C01814=1058.438,-41.200,-66.868,171.247,28.098,155.263
C01815=1058.445,-40.951,-66.880,171.248,28.101,155.263
C01816=1058.451,-40.701,-66.893,171.250,28.102,155.263
C01817=1058.457,-40.452,-66.906,171.252,28.105,155.263
C01818=1058.463,-40.202,-66.919,171.253,28.106,155.264
C01819=1058.469,-39.952,-66.931,171.255,28.108,155.264
C01820=1058.476,-39.703,-66.944,171.257,28.110,155.264
C01821=1058.482,-39.453,-66.956,171.259,28.112,155.264
C01822=1058.488,-39.204,-66.970,171.260,28.114,155.264
C01823=1058.494,-38.954,-66.982,171.262,28.116,155.265
C01824=1058.500,-38.705,-66.996,171.264,28.117,155.265
C01825=1058.507,-38.454,-67.008,171.265,28.120,155.265
C01826=1058.513,-38.205,-67.022,171.267,28.121,155.265
C01827=1058.519,-37.955,-67.034,171.269,28.124,155.265
C01828=1058.525,-37.706,-67.048,171.270,28.126,155.266
C01829=1058.531,-37.456,-67.060,171.272,28.128,155.266
C01830=1058.537,-37.207,-67.073,171.274,28.130,155.266
C01831=1058.543,-36.957,-67.086,171.275,28.131,155.266
C01832=1058.550,-36.708,-67.099,171.277,28.134,155.266
C01833=1058.555,-36.458,-67.112,171.279,28.135,155.267
C01834=1058.562,-36.208,-67.125,171.279,28.137,155.267
C01835=1058.568,-35.959,-67.138,171.281,28.139,155.267
C01836=1058.574,-35.709,-67.151,171.283,28.141,155.267
C01837=1058.580,-35.460,-67.164,171.284,28.144,155.268
C01838=1058.586,-35.210,-67.177,171.286,28.145,155.268
C01839=1058.592,-34.961,-67.190,171.288,28.147,155.268
C01840=1058.599,-34.682,-67.204,171.290,28.150,155.268
C01841=1058.606,-34.402,-67.220,171.292,28.152,155.268
C01842=1058.613,-34.123,-67.234,171.294,28.154,155.269
C01843=1058.620,-33.844,-67.249,171.295,28.156,155.269
C01844=1058.626,-33.594,-67.261,171.297,28.158,155.269
C01845=1058.632,-33.345,-67.275,171.299,28.160,155.269
C01846=1058.638,-33.096,-67.288,171.301,28.162,155.270
C01847=1058.644,-32.846,-67.300,171.302,28.164,155.270
C01848=1058.650,-32.597,-67.314,171.304,28.166,155.270
C01849=1058.656,-32.346,-67.328,171.306,28.168,155.270
C01850=1058.663,-32.097,-67.341,171.307,28.171,155.271
C01851=1058.669,-31.847,-67.354,171.309,28.172,155.271
C01852=1058.675,-31.598,-67.367,171.311,28.175,155.271
C01853=1058.681,-31.349,-67.380,171.312,28.176,155.271
C01854=1058.687,-31.099,-67.393,171.314,28.178,155.271
C01855=1058.694,-30.849,-67.406,171.316,28.181,155.272
C01856=1058.700,-30.600,-67.420,171.317,28.182,155.272
C01857=1058.706,-30.350,-67.433,171.319,28.185,155.272
C01858=1058.712,-30.101,-67.446,171.321,28.186,155.272
C01859=1058.718,-29.851,-67.459,171.322,28.188,155.272
C01860=1058.724,-29.602,-67.473,171.324,28.191,155.273
C01861=1058.731,-29.352,-67.486,171.326,28.192,155.273
C01862=1058.736,-29.102,-67.499,171.327,28.195,155.273
C01863=1058.743,-28.853,-67.512,171.328,28.197,155.273
C01864=1058.749,-28.603,-67.525,171.330,28.198,155.274
C01865=1058.756,-28.353,-67.539,171.331,28.201,155.274
C01866=1058.762,-28.104,-67.552,171.333,28.203,155.274
C01867=1058.768,-27.855,-67.566,171.335,28.204,155.274
C01868=1058.774,-27.605,-67.578,171.337,28.207,155.275
C01869=1058.780,-27.355,-67.592,171.338,28.209,155.275
C01870=1058.786,-27.105,-67.606,171.340,28.211,155.275
C01871=1058.793,-26.856,-67.619,171.342,28.213,155.275
C01872=1058.799,-26.607,-67.632,171.343,28.215,155.275
C01873=1058.805,-26.358,-67.645,171.345,28.217,155.276
C01874=1058.811,-26.107,-67.660,171.347,28.219,155.276
C01875=1058.817,-25.857,-67.672,171.348,28.221,155.276
C01876=1058.823,-25.608,-67.686,171.350,28.223,155.276
C01877=1058.829,-25.359,-67.699,171.352,28.226,155.277
C01878=1058.835,-25.109,-67.713,171.353,28.227,155.277
C01879=1058.842,-24.859,-67.726,171.355,28.230,155.277
C01880=1058.847,-24.610,-67.740,171.357,28.232,155.277
C01881=1058.853,-24.361,-67.753,171.358,28.234,155.278
C01882=1058.860,-24.111,-67.767,171.360,28.236,155.278
C01883=1058.866,-23.861,-67.781,171.362,28.238,155.278
C01884=1058.872,-23.612,-67.794,171.362,28.240,155.278
C01885=1058.877,-23.362,-67.808,171.364,28.242,155.279
C01886=1058.884,-23.113,-67.821,171.366,28.244,155.279
C01887=1058.890,-22.863,-67.835,171.367,28.247,155.279
C01888=1058.896,-22.613,-67.849,171.369,28.249,155.279
C01889=1058.902,-22.364,-67.862,171.371,28.251,155.280
C01890=1058.908,-22.115,-67.875,171.372,28.253,155.280
C01891=1058.914,-21.865,-67.890,171.374,28.255,155.280
C01892=1058.921,-21.615,-67.903,171.376,28.257,155.280
C01893=1058.927,-21.366,-67.916,171.377,28.260,155.281
C01894=1058.933,-21.116,-67.930,171.379,28.261,155.281
C01895=1058.939,-20.867,-67.944,171.381,28.263,155.281
C01896=1058.945,-20.617,-67.957,171.382,28.266,155.281
C01897=1058.951,-20.368,-67.971,171.384,28.268,155.282
C01898=1058.958,-20.118,-67.984,171.386,28.270,155.282
C01899=1058.963,-19.869,-67.999,171.386,28.272,155.282
C01900=1058.970,-19.619,-68.012,171.388,28.274,155.282
C01901=1058.976,-19.370,-68.026,171.390,28.276,155.283
C01902=1058.982,-19.120,-68.040,171.391,28.278,155.283
C01903=1058.988,-18.871,-68.053,171.393,28.281,155.283
C01904=1058.994,-18.590,-68.068,171.395,28.283,155.283
C01905=1059.002,-18.311,-68.084,171.397,28.286,155.284
C01906=1059.009,-18.031,-68.099,171.399,28.288,155.284
C01907=1059.015,-17.751,-68.115,171.401,28.290,155.284
C01908=1059.022,-17.501,-68.128,171.402,28.293,155.285
C01909=1059.028,-17.252,-68.143,171.404,28.295,155.285
C01910=1059.034,-17.003,-68.156,171.406,28.297,155.285
C01911=1059.040,-16.753,-68.170,171.407,28.299,155.285
C01912=1059.047,-16.503,-68.184,171.409,28.301,155.286
C01913=1059.053,-16.253,-68.197,171.410,28.303,155.286
C01914=1059.059,-16.004,-68.211,171.411,28.305,155.286
C01915=1059.065,-15.755,-68.225,171.413,28.307,155.286
C01916=1059.071,-15.505,-68.239,171.415,28.310,155.287
C01917=1059.078,-15.256,-68.253,171.416,28.312,155.287
C01918=1059.084,-15.005,-68.267,171.418,28.314,155.287
C01919=1059.090,-14.757,-68.281,171.420,28.316,155.287
C01920=1059.096,-14.507,-68.295,171.421,28.319,155.288
C01921=1059.103,-14.257,-68.308,171.423,28.321,155.288
C01922=1059.108,-14.008,-68.323,171.425,28.323,155.288
C01923=1059.114,-13.759,-68.337,171.426,28.325,155.289
C01924=1059.121,-13.509,-68.350,171.428,28.328,155.289
C01925=1059.126,-13.259,-68.364,171.429,28.330,155.289
C01926=1059.133,-13.009,-68.379,171.430,28.332,155.289
C01927=1059.139,-12.760,-68.393,171.432,28.334,155.290
C01928=1059.144,-12.511,-68.406,171.434,28.336,155.290
C01929=1059.151,-12.261,-68.421,171.435,28.339,155.290
C01930=1059.157,-12.012,-68.435,171.437,28.341,155.290
C01931=1059.163,-11.761,-68.449,171.439,28.343,155.291
C01932=1059.169,-11.513,-68.463,171.440,28.345,155.291
C01933=1059.175,-11.263,-68.477,171.442,28.347,155.291
C01934=1059.181,-11.013,-68.492,171.443,28.350,155.292
C01935=1059.187,-10.764,-68.505,171.445,28.352,155.292
C01936=1059.194,-10.514,-68.519,171.446,28.354,155.292
C01937=1059.199,-10.265,-68.534,171.448,28.356,155.292
C01938=1059.206,-10.015,-68.547,171.449,28.358,155.293
C01939=1059.212,-9.766,-68.562,171.451,28.361,155.293
C01940=1059.218,-9.516,-68.576,171.453,28.363,155.293
C01941=1059.224,-9.266,-68.589,171.454,28.365,155.293
C01942=1059.231,-9.017,-68.604,171.456,28.367,155.294
C01943=1059.236,-8.767,-68.618,171.457,28.370,155.294
C01944=1059.243,-8.519,-68.632,171.459,28.372,155.294
C01945=1059.249,-8.268,-68.647,171.461,28.374,155.295
C01946=1059.254,-8.019,-68.661,171.462,28.376,155.295
C01947=1059.261,-7.769,-68.675,171.463,28.378,155.295
C01948=1059.267,-7.520,-68.689,171.465,28.381,155.295
C01949=1059.273,-7.270,-68.704,171.467,28.383,155.296
C01950=1059.279,-7.021,-68.718,171.468,28.386,155.296
C01951=1059.286,-6.771,-68.732,171.470,28.388,155.296
C01952=1059.292,-6.522,-68.746,171.471,28.390,155.297
C01953=1059.298,-6.272,-68.761,171.473,28.392,155.297
C01954=1059.304,-6.023,-68.775,171.475,28.394,155.297
C01955=1059.310,-5.773,-68.789,171.476,28.397,155.297
C01956=1059.317,-5.523,-68.804,171.477,28.399,155.298
C01957=1059.322,-5.274,-68.818,171.479,28.401,155.298
C01958=1059.329,-5.025,-68.832,171.480,28.403,155.298
C01959=1059.335,-4.776,-68.847,171.482,28.405,155.298
C01960=1059.341,-4.525,-68.861,171.484,28.408,155.299
C01961=1059.348,-4.277,-68.875,171.485,28.410,155.299
C01962=1059.354,-4.026,-68.889,171.487,28.412,155.299
C01963=1059.359,-3.777,-68.904,171.489,28.414,155.300
C01964=1059.366,-3.528,-68.918,171.490,28.417,155.300
C01965=1059.373,-3.278,-68.932,171.491,28.419,155.300
C01966=1059.378,-3.029,-68.947,171.493,28.421,155.301
C01967=1059.384,-2.779,-68.961,171.494,28.424,155.301
C01968=1059.391,-2.498,-68.978,171.496,28.426,155.301
C01969=1059.397,-2.216,-68.994,171.498,28.429,155.301
C01970=1059.405,-1.935,-69.010,171.500,28.432,155.302
C01971=1059.411,-1.653,-69.027,171.502,28.435,155.302
C01972=1059.417,-1.403,-69.042,171.503,28.437,155.302
C01973=1059.423,-1.154,-69.056,171.504,28.439,155.303
C01974=1059.429,-0.904,-69.071,171.506,28.441,155.303
C01975=1059.435,-0.655,-69.085,171.507,28.444,155.303
C01976=1059.441,-0.406,-69.100,171.509,28.446,155.304
C01977=1059.447,-0.157,-69.115,171.511,28.448,155.304
C01978=1059.453,0.094,-69.129,171.512,28.450,155.304
C01979=1059.459,0.343,-69.143,171.514,28.453,155.305
C01980=1059.465,0.592,-69.158,171.516,28.456,155.305
C01981=1059.472,0.842,-69.173,171.516,28.458,155.305
C01982=1059.477,1.092,-69.187,171.518,28.460,155.305
C01983=1059.484,1.341,-69.202,171.520,28.463,155.306
C01984=1059.489,1.590,-69.217,171.521,28.465,155.306
C01985=1059.496,1.840,-69.232,171.523,28.467,155.306
C01986=1059.501,2.089,-69.246,171.525,28.469,155.307
C01987=1059.508,2.339,-69.260,171.526,28.472,155.307
C01988=1059.514,2.589,-69.275,171.527,28.474,155.307
C01989=1059.520,2.838,-69.290,171.529,28.476,155.308
C01990=1059.526,3.087,-69.305,171.530,28.478,155.308
C01991=1059.532,3.337,-69.320,171.532,28.481,155.308
C01992=1059.538,3.586,-69.334,171.534,28.484,155.309
C01993=1059.544,3.836,-69.349,171.535,28.486,155.309
C01994=1059.550,4.085,-69.363,171.537,28.489,155.309
C01995=1059.557,4.335,-69.378,171.538,28.491,155.309
C01996=1059.563,4.584,-69.393,171.539,28.493,155.310
C01997=1059.569,4.833,-69.408,171.541,28.495,155.310
C01998=1059.574,5.083,-69.423,171.542,28.498,155.310
C01999=1059.581,5.333,-69.438,171.544,28.500,155.311
C02000=1059.586,5.582,-69.453,171.546,28.502,155.311
C02001=1059.593,5.832,-69.468,171.547,28.504,155.311
C02002=1059.599,6.081,-69.483,171.549,28.507,155.312
C02003=1059.605,6.331,-69.497,171.550,28.509,155.312
C02004=1059.611,6.581,-69.512,171.551,28.512,155.312
C02005=1059.618,6.830,-69.526,171.553,28.514,155.313
C02006=1059.623,7.079,-69.541,171.555,28.517,155.313
C02007=1059.630,7.329,-69.556,171.556,28.519,155.313
C02008=1059.636,7.578,-69.571,171.558,28.521,155.313
C02009=1059.642,7.827,-69.586,171.560,28.524,155.314
C02010=1059.648,8.077,-69.600,171.560,28.526,155.314
C02011=1059.654,8.327,-69.616,171.562,28.528,155.314
C02012=1059.660,8.577,-69.631,171.564,28.530,155.315
C02013=1059.666,8.826,-69.646,171.565,28.533,155.315
C02014=1059.672,9.075,-69.660,171.567,28.535,155.315
C02015=1059.679,9.325,-69.675,171.569,28.537,155.316
C02016=1059.685,9.574,-69.690,171.570,28.540,155.316
C02017=1059.691,9.824,-69.705,171.571,28.542,155.316
C02018=1059.697,10.073,-69.720,171.573,28.544,155.317
C02019=1059.704,10.322,-69.736,171.574,28.547,155.317
C02020=1059.710,10.571,-69.750,171.576,28.550,155.317
C02021=1059.715,10.821,-69.766,171.578,28.552,155.318
C02022=1059.722,11.071,-69.781,171.579,28.554,155.318
C02023=1059.728,11.320,-69.796,171.581,28.556,155.318
C02024=1059.735,11.570,-69.811,171.582,28.559,155.318
C02025=1059.740,11.819,-69.825,171.583,28.561,155.319
C02026=1059.747,12.069,-69.840,171.585,28.563,155.319
C02027=1059.753,12.318,-69.855,171.587,28.566,155.319
C02028=1059.760,12.568,-69.870,171.588,28.568,155.320
C02029=1059.765,12.817,-69.886,171.590,28.570,155.320
C02030=1059.771,13.066,-69.901,171.592,28.573,155.320
C02031=1059.778,13.316,-69.916,171.592,28.575,155.321
C02032=1059.785,13.600,-69.932,171.595,28.578,155.321
C02033=1059.792,13.883,-69.950,171.596,28.580,155.321
C02034=1059.799,14.166,-69.967,171.598,28.583,155.322
C02035=1059.806,14.450,-69.984,171.600,28.586,155.322
C02036=1059.812,14.699,-70.000,171.601,28.588,155.322
C02037=1059.819,14.949,-70.015,171.603,28.591,155.323
C02038=1059.824,15.198,-70.030,171.604,28.593,155.323
C02039=1059.830,15.448,-70.045,171.605,28.595,155.323
C02040=1059.837,15.697,-70.060,171.607,28.598,155.324
C02041=1059.843,15.947,-70.076,171.609,28.600,155.324
C02042=1059.848,16.196,-70.091,171.610,28.603,155.324
C02043=1059.854,16.446,-70.106,171.612,28.605,155.325
C02044=1059.860,16.695,-70.121,171.613,28.607,155.325
C02045=1059.867,16.944,-70.137,171.614,28.610,155.325
C02046=1059.873,17.194,-70.152,171.616,28.612,155.326
C02047=1059.878,17.443,-70.167,171.617,28.615,155.326
C02048=1059.885,17.692,-70.183,171.619,28.617,155.326
C02049=1059.891,17.942,-70.198,171.621,28.620,155.327
C02050=1059.897,18.192,-70.213,171.622,28.622,155.327
C02051=1059.904,18.441,-70.229,171.623,28.624,155.327
C02052=1059.910,18.691,-70.244,171.625,28.627,155.328
C02053=1059.915,18.940,-70.259,171.626,28.629,155.328
C02054=1059.921,19.189,-70.275,171.628,28.632,155.328
C02055=1059.928,19.439,-70.290,171.630,28.634,155.329
C02056=1059.934,19.688,-70.305,171.630,28.636,155.329
C02057=1059.940,19.938,-70.321,171.632,28.639,155.329
C02058=1059.946,20.187,-70.336,171.634,28.641,155.330
C02059=1059.952,20.437,-70.352,171.635,28.644,155.330
C02060=1059.958,20.686,-70.367,171.637,28.646,155.330
C02061=1059.964,20.936,-70.383,171.639,28.649,155.331
C02062=1059.970,21.185,-70.398,171.639,28.651,155.331
C02063=1059.976,21.435,-70.414,171.641,28.654,155.331
C02064=1059.983,21.684,-70.429,171.643,28.656,155.332
C02065=1059.988,21.934,-70.445,171.644,28.659,155.332
C02066=1059.995,22.183,-70.461,171.646,28.661,155.332
C02067=1060.000,22.432,-70.476,171.648,28.664,155.333
C02068=1060.007,22.682,-70.491,171.648,28.666,155.333
C02069=1060.012,22.931,-70.507,171.650,28.669,155.333
C02070=1060.019,23.181,-70.522,171.652,28.671,155.334
C02071=1060.025,23.430,-70.538,171.653,28.673,155.334
C02072=1060.031,23.680,-70.553,171.655,28.676,155.334
C02073=1060.037,23.929,-70.569,171.656,28.678,155.335
C02074=1060.044,24.179,-70.584,171.657,28.681,155.335
C02075=1060.049,24.428,-70.601,171.659,28.683,155.335
C02076=1060.056,24.678,-70.616,171.661,28.686,155.336
C02077=1060.061,24.926,-70.631,171.662,28.688,155.336
C02078=1060.067,25.176,-70.648,171.664,28.691,155.336
C02079=1060.074,25.425,-70.663,171.665,28.693,155.337
C02080=1060.079,25.675,-70.679,171.666,28.696,155.337
C02081=1060.086,25.924,-70.694,171.668,28.698,155.337
C02082=1060.092,26.174,-70.710,171.669,28.701,155.338
C02083=1060.098,26.423,-70.725,171.671,28.703,155.338
C02084=1060.104,26.673,-70.741,171.673,28.706,155.338
C02085=1060.111,26.922,-70.757,171.673,28.708,155.339
C02086=1060.116,27.172,-70.773,171.675,28.710,155.339
C02087=1060.122,27.421,-70.789,171.677,28.713,155.339
C02088=1060.129,27.671,-70.804,171.678,28.715,155.340
C02089=1060.135,27.920,-70.820,171.680,28.718,155.340
C02090=1060.141,28.169,-70.836,171.682,28.720,155.340
C02091=1060.147,28.419,-70.851,171.682,28.722,155.341
C02092=1060.153,28.668,-70.867,171.684,28.725,155.341
C02093=1060.160,28.918,-70.883,171.686,28.727,155.341
C02094=1060.165,29.167,-70.899,171.687,28.730,155.342
C02095=1060.171,29.417,-70.915,171.689,28.733,155.342
C02096=1060.178,29.701,-70.932,171.691,28.736,155.342
C02097=1060.185,29.986,-70.951,171.692,28.739,155.343
C02098=1060.192,30.271,-70.969,171.694,28.741,155.343
C02099=1060.199,30.555,-70.987,171.695,28.744,155.344
C02100=1060.204,30.805,-71.003,171.697,28.746,155.344
C02101=1060.210,31.054,-71.019,171.698,28.749,155.344
C02102=1060.216,31.304,-71.035,171.699,28.752,155.345
C02103=1060.223,31.553,-71.051,171.701,28.754,155.345
C02104=1060.229,31.803,-71.066,171.703,28.757,155.345
C02105=1060.235,32.052,-71.083,171.704,28.759,155.346
C02106=1060.241,32.301,-71.099,171.706,28.762,155.346
C02107=1060.247,32.550,-71.115,171.707,28.764,155.347
C02108=1060.253,32.800,-71.131,171.708,28.766,155.347
C02109=1060.259,33.050,-71.146,171.710,28.769,155.347
C02110=1060.265,33.299,-71.163,171.712,28.771,155.347
C02111=1060.272,33.548,-71.178,171.713,28.774,155.348
C02112=1060.277,33.797,-71.195,171.714,28.776,155.348
C02113=1060.283,34.047,-71.211,171.716,28.779,155.349
C02114=1060.289,34.296,-71.227,171.717,28.782,155.349
C02115=1060.296,34.547,-71.243,171.719,28.784,155.349
C02116=1060.302,34.796,-71.259,171.721,28.787,155.350
C02117=1060.308,35.045,-71.275,171.722,28.789,155.350
C02118=1060.314,35.294,-71.291,171.723,28.792,155.350
C02119=1060.320,35.544,-71.307,171.725,28.794,155.351
C02120=1060.326,35.793,-71.324,171.726,28.797,155.351
C02121=1060.333,36.042,-71.339,171.728,28.799,155.351
C02122=1060.339,36.292,-71.356,171.729,28.801,155.352
C02123=1060.344,36.542,-71.371,171.730,28.804,155.352
C02124=1060.350,36.791,-71.387,171.732,28.806,155.352
C02125=1060.356,37.040,-71.404,171.733,28.809,155.353
C02126=1060.363,37.289,-71.419,171.735,28.811,155.353
C02127=1060.369,37.539,-71.436,171.737,28.814,155.353
C02128=1060.376,37.789,-71.452,171.738,28.816,155.354
C02129=1060.381,38.038,-71.468,171.739,28.819,155.354
C02130=1060.387,38.287,-71.485,171.741,28.822,155.355
C02131=1060.393,38.537,-71.501,171.742,28.824,155.355
C02132=1060.399,38.786,-71.517,171.744,28.827,155.355
C02133=1060.405,39.035,-71.533,171.745,28.829,155.356
C02134=1060.411,39.285,-71.550,171.746,28.832,155.356
C02135=1060.417,39.534,-71.566,171.748,28.834,155.356
C02136=1060.423,39.783,-71.582,171.750,28.837,155.357
C02137=1060.429,40.033,-71.598,171.751,28.840,155.357
C02138=1060.435,40.282,-71.615,171.752,28.842,155.357
C02139=1060.441,40.532,-71.631,171.754,28.844,155.358
C02140=1060.448,40.782,-71.648,171.755,28.847,155.358
C02141=1060.453,41.031,-71.664,171.757,28.849,155.358
C02142=1060.459,41.280,-71.680,171.759,28.852,155.359
C02143=1060.465,41.530,-71.696,171.760,28.854,155.359
C02144=1060.472,41.778,-71.713,171.761,28.857,155.360
C02145=1060.478,42.028,-71.730,171.763,28.860,155.360
C02146=1060.484,42.277,-71.746,171.764,28.862,155.360
C02147=1060.489,42.526,-71.762,171.766,28.865,155.361
C02148=1060.496,42.776,-71.779,171.768,28.867,155.361
C02149=1060.502,43.026,-71.795,171.768,28.869,155.361
C02150=1060.508,43.275,-71.811,171.770,28.872,155.362
C02151=1060.514,43.524,-71.827,171.772,28.875,155.362
C02152=1060.520,43.774,-71.844,171.773,28.877,155.362
C02153=1060.525,44.023,-71.861,171.775,28.880,155.363
C02154=1060.531,44.272,-71.878,171.776,28.883,155.363
C02155=1060.538,44.522,-71.894,171.777,28.885,155.364
C02156=1060.544,44.772,-71.910,171.779,28.888,155.364
C02157=1060.549,45.021,-71.927,171.780,28.890,155.364
C02158=1060.555,45.270,-71.944,171.782,28.893,155.365
C02159=1060.561,45.519,-71.961,171.783,28.896,155.365
C02160=1060.568,45.804,-71.980,171.784,28.898,155.365
C02161=1060.574,46.089,-71.999,171.786,28.901,155.366
C02162=1060.581,46.374,-72.018,171.788,28.905,155.366
C02163=1060.588,46.659,-72.037,171.789,28.907,155.367
C02164=1060.594,46.908,-72.053,171.791,28.910,155.367
C02165=1060.600,47.157,-72.069,171.792,28.913,155.368
C02166=1060.606,47.406,-72.087,171.794,28.915,155.368
C02167=1060.612,47.656,-72.103,171.796,28.918,155.368
C02168=1060.618,47.905,-72.119,171.796,28.920,155.369
C02169=1060.624,48.155,-72.137,171.798,28.923,155.369
C02170=1060.630,48.404,-72.153,171.800,28.925,155.369
C02171=1060.636,48.653,-72.170,171.801,28.928,155.370
C02172=1060.642,48.902,-72.187,171.803,28.931,155.370
C02173=1060.647,49.152,-72.204,171.804,28.934,155.371
C02174=1060.653,49.401,-72.220,171.805,28.936,155.371
C02175=1060.660,49.651,-72.237,171.807,28.938,155.371
C02176=1060.665,49.900,-72.254,171.809,28.941,155.372
C02177=1060.671,50.150,-72.270,171.810,28.944,155.372
C02178=1060.677,50.398,-72.287,171.811,28.946,155.372
C02179=1060.684,50.648,-72.304,171.813,28.949,155.373
C02180=1060.689,50.898,-72.321,171.814,28.952,155.373
C02181=1060.695,51.147,-72.338,171.816,28.954,155.374
C02182=1060.701,51.396,-72.354,171.818,28.957,155.374
C02183=1060.707,51.646,-72.372,171.818,28.959,155.374
C02184=1060.713,51.895,-72.388,171.820,28.962,155.375
C02185=1060.719,52.145,-72.404,171.822,28.965,155.375
C02186=1060.725,52.394,-72.422,171.823,28.967,155.375
C02187=1060.731,52.644,-72.439,171.825,28.970,155.376
C02188=1060.738,52.892,-72.456,171.826,28.972,155.376
C02189=1060.743,53.142,-72.472,171.827,28.975,155.377
C02190=1060.749,53.391,-72.489,171.829,28.977,155.377
C02191=1060.756,53.641,-72.506,171.831,28.980,155.377
C02192=1060.762,53.890,-72.523,171.832,28.983,155.378
C02193=1060.767,54.139,-72.540,171.833,28.985,155.378
C02194=1060.773,54.388,-72.557,171.835,28.987,155.378
C02195=1060.780,54.638,-72.573,171.836,28.990,155.379
C02196=1060.785,54.887,-72.591,171.838,28.993,155.379
C02197=1060.791,55.136,-72.607,171.840,28.996,155.379
C02198=1060.798,55.386,-72.625,171.840,28.998,155.380
C02199=1060.804,55.635,-72.641,171.842,29.000,155.380
C02200=1060.810,55.884,-72.658,171.844,29.003,155.381
C02201=1060.816,56.135,-72.676,171.845,29.005,155.381
C02202=1060.822,56.383,-72.693,171.847,29.008,155.381
C02203=1060.828,56.633,-72.709,171.848,29.011,155.382
C02204=1060.834,56.882,-72.727,171.849,29.013,155.382
C02205=1060.840,57.131,-72.744,171.851,29.016,155.382
C02206=1060.846,57.380,-72.760,171.853,29.018,155.383
C02207=1060.852,57.630,-72.778,171.854,29.021,155.383
C02208=1060.858,57.880,-72.794,171.855,29.023,155.383
C02209=1060.864,58.128,-72.811,171.857,29.026,155.384
C02210=1060.871,58.378,-72.829,171.858,29.029,155.384
C02211=1060.877,58.627,-72.845,171.860,29.031,155.385
C02212=1060.883,58.877,-72.863,171.862,29.034,155.385
C02213=1060.889,59.126,-72.880,171.862,29.036,155.385
C02214=1060.895,59.375,-72.897,171.864,29.039,155.386
C02215=1060.901,59.625,-72.914,171.866,29.041,155.386
C02216=1060.907,59.874,-72.931,171.867,29.044,155.386
C02217=1060.914,60.124,-72.948,171.869,29.047,155.387
C02218=1060.919,60.373,-72.966,171.870,29.049,155.387
C02219=1060.926,60.621,-72.983,171.871,29.051,155.388
C02220=1060.931,60.872,-73.000,171.873,29.054,155.388
C02221=1060.938,61.121,-73.017,171.875,29.057,155.388
C02222=1060.944,61.370,-73.034,171.876,29.059,155.389
C02223=1060.950,61.620,-73.051,171.878,29.062,155.389
C02224=1060.957,61.904,-73.071,171.880,29.065,155.389
C02225=1060.965,62.188,-73.090,171.881,29.067,155.390
C02226=1060.971,62.473,-73.110,171.883,29.070,155.390
C02227=1060.978,62.757,-73.129,171.884,29.074,155.391
C02228=1060.985,63.006,-73.147,171.886,29.076,155.391
C02229=1060.990,63.255,-73.164,171.887,29.078,155.391
C02230=1060.997,63.505,-73.182,171.888,29.081,155.392
C02231=1061.002,63.755,-73.198,171.890,29.083,155.392
C02232=1061.009,64.004,-73.216,171.892,29.086,155.393
C02233=1061.015,64.253,-73.233,171.893,29.089,155.393
C02234=1061.021,64.502,-73.251,171.894,29.091,155.393
C02235=1061.027,64.751,-73.268,171.896,29.093,155.394
C02236=1061.033,65.002,-73.285,171.898,29.096,155.394
C02237=1061.039,65.251,-73.302,171.899,29.099,155.394
C02238=1061.044,65.500,-73.320,171.901,29.102,155.395
C02239=1061.051,65.749,-73.337,171.902,29.104,155.395
C02240=1061.057,65.998,-73.355,171.903,29.106,155.396
C02241=1061.063,66.248,-73.373,171.905,29.109,155.396
C02242=1061.069,66.497,-73.390,171.907,29.112,155.396
C02243=1061.075,66.747,-73.407,171.908,29.115,155.397
C02244=1061.081,66.996,-73.425,171.909,29.117,155.397
C02245=1061.087,67.245,-73.442,171.911,29.119,155.397
C02246=1061.093,67.494,-73.459,171.912,29.122,155.398
C02247=1061.099,67.744,-73.477,171.914,29.125,155.398
C02248=1061.105,67.993,-73.494,171.916,29.128,155.399
C02249=1061.111,68.243,-73.512,171.916,29.130,155.399
C02250=1061.117,68.492,-73.530,171.918,29.132,155.399
C02251=1061.123,68.740,-73.547,171.920,29.135,155.400
C02252=1061.129,68.990,-73.565,171.921,29.138,155.400
C02253=1061.135,69.239,-73.582,171.923,29.141,155.401
C02254=1061.141,69.489,-73.600,171.924,29.143,155.401
C02255=1061.147,69.738,-73.617,171.925,29.145,155.401
C02256=1061.153,69.987,-73.635,171.927,29.148,155.402
C02257=1061.159,70.236,-73.653,171.929,29.151,155.402
C02258=1061.165,70.486,-73.671,171.930,29.154,155.402
C02259=1061.171,70.735,-73.688,171.931,29.156,155.403
C02260=1061.177,70.985,-73.706,171.933,29.158,155.403
C02261=1061.183,71.234,-73.723,171.934,29.161,155.404
C02262=1061.189,71.483,-73.741,171.936,29.164,155.404
C02263=1061.195,71.732,-73.759,171.938,29.167,155.404
C02264=1061.201,71.982,-73.777,171.939,29.169,155.405
C02265=1061.206,72.231,-73.794,171.940,29.172,155.405
C02266=1061.213,72.481,-73.811,171.942,29.175,155.406
C02267=1061.219,72.730,-73.830,171.943,29.177,155.406
C02268=1061.225,72.979,-73.848,171.945,29.180,155.406
C02269=1061.231,73.229,-73.866,171.947,29.182,155.407
C02270=1061.237,73.478,-73.883,171.947,29.185,155.407
C02271=1061.243,73.727,-73.901,171.949,29.188,155.407
C02272=1061.248,73.976,-73.919,171.951,29.191,155.408
C02273=1061.254,74.226,-73.937,171.952,29.193,155.408
C02274=1061.261,74.475,-73.954,171.954,29.195,155.409
C02275=1061.267,74.724,-73.972,171.955,29.198,155.409
C02276=1061.273,74.973,-73.990,171.956,29.201,155.409
C02277=1061.279,75.223,-74.008,171.958,29.203,155.410
C02278=1061.285,75.473,-74.026,171.960,29.206,155.410
C02279=1061.290,75.722,-74.043,171.961,29.208,155.410
C02280=1061.297,75.971,-74.062,171.962,29.211,155.411
C02281=1061.302,76.220,-74.079,171.964,29.214,155.411
C02282=1061.308,76.469,-74.097,171.965,29.216,155.412
C02283=1061.315,76.718,-74.114,171.967,29.219,155.412
C02284=1061.321,76.968,-74.132,171.969,29.221,155.412
C02285=1061.327,77.217,-74.151,171.969,29.224,155.413
C02286=1061.333,77.466,-74.169,171.971,29.227,155.413
C02287=1061.339,77.716,-74.186,171.973,29.229,155.414
C02288=1061.346,78.000,-74.207,171.974,29.232,155.414
C02289=1061.352,78.284,-74.228,171.976,29.236,155.415
C02290=1061.359,78.569,-74.248,171.978,29.238,155.415
C02291=1061.366,78.853,-74.269,171.979,29.242,155.415
C02292=1061.372,79.102,-74.287,171.981,29.244,155.416
C02293=1061.378,79.352,-74.305,171.983,29.247,155.416
C02294=1061.384,79.600,-74.323,171.984,29.249,155.417
C02295=1061.390,79.850,-74.341,171.986,29.252,155.417
C02296=1061.396,80.100,-74.359,171.987,29.255,155.417
C02297=1061.401,80.348,-74.378,171.988,29.257,155.418
C02298=1061.407,80.598,-74.396,171.990,29.260,155.418
C02299=1061.413,80.847,-74.414,171.992,29.263,155.419
C02300=1061.419,81.096,-74.432,171.993,29.266,155.419
C02301=1061.425,81.346,-74.450,171.994,29.268,155.419
C02302=1061.431,81.594,-74.468,171.996,29.271,155.420
C02303=1061.437,81.844,-74.486,171.997,29.274,155.420
C02304=1061.442,82.093,-74.505,171.999,29.276,155.420
C02305=1061.448,82.343,-74.523,172.001,29.278,155.421
C02306=1061.454,82.592,-74.541,172.002,29.281,155.421
C02307=1061.460,82.841,-74.559,172.003,29.284,155.422
C02308=1061.466,83.091,-74.577,172.005,29.287,155.422
C02309=1061.473,83.340,-74.596,172.006,29.289,155.422
C02310=1061.478,83.589,-74.613,172.008,29.292,155.423
C02311=1061.484,83.838,-74.632,172.010,29.295,155.423
C02312=1061.490,84.088,-74.650,172.010,29.297,155.424
C02313=1061.496,84.336,-74.669,172.012,29.299,155.424
C02314=1061.502,84.586,-74.686,172.014,29.302,155.424
C02315=1061.508,84.835,-74.705,172.016,29.305,155.425
C02316=1061.514,85.084,-74.723,172.017,29.308,155.425
C02317=1061.520,85.334,-74.742,172.019,29.310,155.426
C02318=1061.526,85.583,-74.760,172.020,29.313,155.426
C02319=1061.532,85.832,-74.778,172.021,29.316,155.426
C02320=1061.538,86.082,-74.796,172.023,29.318,155.427
C02321=1061.544,86.331,-74.815,172.025,29.321,155.427
C02322=1061.550,86.581,-74.833,172.026,29.323,155.428
C02323=1061.555,86.829,-74.852,172.028,29.326,155.428
C02324=1061.562,87.078,-74.870,172.029,29.329,155.428
C02325=1061.568,87.328,-74.888,172.030,29.331,155.429
C02326=1061.574,87.577,-74.907,172.032,29.334,155.429
C02327=1061.580,87.826,-74.924,172.034,29.337,155.430
C02328=1061.586,88.076,-74.944,172.035,29.339,155.430
C02329=1061.592,88.325,-74.962,172.036,29.342,155.430
C02330=1061.598,88.574,-74.980,172.038,29.344,155.431
C02331=1061.604,88.823,-74.998,172.039,29.347,155.431
C02332=1061.610,89.073,-75.016,172.041,29.350,155.431
C02333=1061.616,89.322,-75.036,172.043,29.353,155.432
C02334=1061.622,89.571,-75.054,172.045,29.355,155.432
C02335=1061.628,89.820,-75.072,172.045,29.357,155.433
C02336=1061.634,90.069,-75.090,172.047,29.360,155.433
C02337=1061.640,90.319,-75.110,172.049,29.363,155.433
C02338=1061.646,90.569,-75.128,172.050,29.365,155.434
C02339=1061.652,90.818,-75.146,172.052,29.368,155.434
C02340=1061.657,91.066,-75.165,172.054,29.371,155.435
C02341=1061.664,91.315,-75.184,172.054,29.373,155.435
C02342=1061.670,91.565,-75.202,172.056,29.376,155.435
C02343=1061.675,91.814,-75.221,172.058,29.378,155.436
C02344=1061.681,92.063,-75.239,172.059,29.381,155.436
C02345=1061.687,92.313,-75.259,172.061,29.384,155.437
C02346=1061.693,92.562,-75.276,172.063,29.387,155.437
C02347=1061.699,92.812,-75.296,172.063,29.389,155.437
C02348=1061.705,93.060,-75.314,172.065,29.392,155.438
C02349=1061.710,93.310,-75.333,172.067,29.395,155.438
C02350=1061.717,93.559,-75.352,172.068,29.397,155.439
C02351=1061.723,93.808,-75.370,172.070,29.400,155.439
C02352=1061.729,94.093,-75.391,172.072,29.403,155.439
C02353=1061.736,94.377,-75.412,172.073,29.406,155.440
C02354=1061.742,94.661,-75.434,172.075,29.409,155.440
C02355=1061.749,94.945,-75.455,172.077,29.412,155.441
C02356=1061.755,95.194,-75.474,172.078,29.415,155.441
C02357=1061.762,95.443,-75.493,172.080,29.418,155.442
C02358=1061.767,95.693,-75.512,172.082,29.420,155.442
C02359=1061.774,95.942,-75.531,172.083,29.423,155.442
C02360=1061.779,96.191,-75.550,172.084,29.426,155.443
C02361=1061.785,96.440,-75.568,172.086,29.428,155.443
C02362=1061.791,96.690,-75.587,172.088,29.431,155.444
C02363=1061.797,96.939,-75.606,172.089,29.433,155.444
C02364=1061.803,97.188,-75.625,172.091,29.436,155.444
C02365=1061.809,97.438,-75.643,172.093,29.439,155.445
C02366=1061.815,97.687,-75.663,172.093,29.441,155.445
C02367=1061.821,97.936,-75.681,172.095,29.444,155.446
C02368=1061.826,98.185,-75.700,172.097,29.447,155.446
C02369=1061.833,98.434,-75.719,172.098,29.449,155.446
C02370=1061.838,98.683,-75.738,172.100,29.452,155.447
C02371=1061.845,98.933,-75.757,172.102,29.454,155.447
C02372=1061.851,99.182,-75.776,172.103,29.457,155.447
C02373=1061.857,99.431,-75.795,172.104,29.460,155.448
C02374=1061.863,99.681,-75.814,172.106,29.462,155.448
C02375=1061.869,99.930,-75.833,172.107,29.465,155.449
C02376=1061.875,100.179,-75.852,172.109,29.468,155.449
C02377=1061.881,100.428,-75.870,172.111,29.471,155.450
C02378=1061.886,100.677,-75.889,172.113,29.473,155.450
C02379=1061.893,100.926,-75.908,172.114,29.475,155.450
C02380=1061.898,101.176,-75.927,172.115,29.478,155.451
C02381=1061.904,101.425,-75.946,172.117,29.481,155.451
C02382=1061.910,101.674,-75.966,172.118,29.483,155.451
C02383=1061.916,101.923,-75.984,172.120,29.486,155.452
C02384=1061.922,102.173,-76.004,172.122,29.489,155.452
C02385=1061.928,102.422,-76.024,172.123,29.492,155.453
C02386=1061.934,102.671,-76.043,172.125,29.494,155.453
C02387=1061.939,102.920,-76.061,172.126,29.497,155.453
C02388=1061.945,103.169,-76.080,172.127,29.500,155.454
C02389=1061.951,103.418,-76.100,172.129,29.502,155.454
C02390=1061.956,103.668,-76.119,172.131,29.505,155.455
C02391=1061.963,103.917,-76.137,172.133,29.508,155.455
C02392=1061.969,104.166,-76.157,172.134,29.510,155.456
C02393=1061.975,104.415,-76.177,172.136,29.513,155.456
C02394=1061.980,104.665,-76.196,172.137,29.516,155.456
C02395=1061.987,104.914,-76.215,172.138,29.518,155.457
C02396=1061.992,105.163,-76.234,172.140,29.521,155.457
C02397=1061.998,105.412,-76.254,172.142,29.524,155.458
C02398=1062.004,105.661,-76.273,172.143,29.527,155.458
C02399=1062.010,105.910,-76.291,172.145,29.529,155.458
C02400=1062.016,106.159,-76.311,172.147,29.532,155.459
C02401=1062.022,106.408,-76.330,172.148,29.535,155.459
C02402=1062.027,106.658,-76.350,172.149,29.537,155.460
C02403=1062.033,106.907,-76.369,172.151,29.540,155.460
C02404=1062.039,107.156,-76.388,172.152,29.543,155.460
C02405=1062.045,107.405,-76.408,172.154,29.545,155.461
C02406=1062.051,107.654,-76.427,172.156,29.548,155.461
C02407=1062.057,107.904,-76.446,172.158,29.551,155.462
C02408=1062.063,108.153,-76.465,172.159,29.553,155.462
C02409=1062.069,108.402,-76.485,172.161,29.556,155.462
C02410=1062.075,108.651,-76.504,172.162,29.558,155.463
C02411=1062.081,108.901,-76.523,172.163,29.561,155.463
C02412=1062.087,109.149,-76.543,172.165,29.564,155.464
C02413=1062.093,109.399,-76.562,172.167,29.566,155.464
C02414=1062.099,109.648,-76.581,172.168,29.569,155.464
C02415=1062.105,109.897,-76.601,172.170,29.572,155.465
C02416=1062.111,110.182,-76.623,172.172,29.575,155.465
C02417=1062.119,110.466,-76.646,172.173,29.578,155.466
C02418=1062.125,110.750,-76.667,172.175,29.581,155.466
C02419=1062.132,111.035,-76.690,172.177,29.584,155.467
C02420=1062.138,111.284,-76.709,172.178,29.587,155.467
C02421=1062.144,111.533,-76.729,172.180,29.589,155.467
C02422=1062.150,111.782,-76.748,172.182,29.592,155.468
C02423=1062.156,112.031,-76.768,172.184,29.595,155.468
C02424=1062.162,112.280,-76.787,172.185,29.598,155.469
C02425=1062.168,112.529,-76.807,172.187,29.600,155.469
C02426=1062.173,112.779,-76.826,172.189,29.602,155.469
C02427=1062.179,113.027,-76.846,172.190,29.605,155.470
C02428=1062.185,113.277,-76.865,172.192,29.608,155.470
C02429=1062.191,113.526,-76.885,172.193,29.610,155.471
C02430=1062.197,113.775,-76.905,172.195,29.613,155.471
C02431=1062.203,114.024,-76.925,172.196,29.616,155.471
C02432=1062.209,114.273,-76.944,172.198,29.619,155.472
C02433=1062.215,114.522,-76.964,172.200,29.621,155.472
C02434=1062.219,114.772,-76.984,172.201,29.624,155.473
C02435=1062.225,115.021,-77.004,172.203,29.627,155.473
C02436=1062.231,115.270,-77.023,172.205,29.630,155.474
C02437=1062.237,115.519,-77.043,172.206,29.633,155.474
C02438=1062.243,115.768,-77.062,172.207,29.635,155.474
C02439=1062.249,116.018,-77.082,172.209,29.638,155.475
C02440=1062.255,116.267,-77.103,172.210,29.641,155.475
C02441=1062.260,116.517,-77.122,172.212,29.643,155.476
C02442=1062.266,116.765,-77.142,172.214,29.646,155.476
C02443=1062.272,117.014,-77.162,172.216,29.649,155.476
C02444=1062.278,117.264,-77.181,172.217,29.652,155.477
C02445=1062.283,117.513,-77.202,172.219,29.654,155.477
C02446=1062.289,117.762,-77.221,172.221,29.657,155.478
C02447=1062.295,118.011,-77.241,172.222,29.660,155.478
C02448=1062.301,118.260,-77.261,172.223,29.662,155.478
C02449=1062.307,118.509,-77.281,172.225,29.665,155.479
C02450=1062.312,118.758,-77.301,172.226,29.668,155.479
C02451=1062.318,119.007,-77.321,172.228,29.671,155.480
C02452=1062.325,119.257,-77.341,172.230,29.674,155.480
C02453=1062.330,119.506,-77.360,172.231,29.676,155.481
C02454=1062.336,119.755,-77.380,172.233,29.679,155.481
C02455=1062.341,120.004,-77.401,172.235,29.682,155.481
C02456=1062.347,120.253,-77.421,172.237,29.685,155.482
C02457=1062.353,120.502,-77.440,172.238,29.687,155.482
C02458=1062.359,120.751,-77.460,172.240,29.690,155.483
C02459=1062.364,121.000,-77.481,172.241,29.692,155.483
C02460=1062.371,121.250,-77.501,172.242,29.695,155.484
C02461=1062.377,121.499,-77.520,172.244,29.698,155.484
C02462=1062.383,121.748,-77.540,172.246,29.701,155.484
C02463=1062.388,121.997,-77.561,172.248,29.703,155.485
C02464=1062.394,122.246,-77.581,172.249,29.706,155.485
C02465=1062.400,122.495,-77.601,172.251,29.709,155.486
C02466=1062.406,122.745,-77.620,172.253,29.711,155.486
C02467=1062.411,122.994,-77.641,172.254,29.714,155.486
C02468=1062.417,123.243,-77.661,172.256,29.717,155.487
C02469=1062.423,123.492,-77.681,172.258,29.720,155.487
C02470=1062.429,123.740,-77.701,172.259,29.722,155.488
C02471=1062.435,123.990,-77.722,172.261,29.725,155.488
C02472=1062.441,124.239,-77.741,172.263,29.728,155.488
C02473=1062.447,124.488,-77.761,172.265,29.730,155.489
C02474=1062.453,124.737,-77.781,172.265,29.733,155.489
C02475=1062.458,124.986,-77.801,172.267,29.736,155.490
C02476=1062.465,125.236,-77.822,172.269,29.738,155.490
C02477=1062.471,125.485,-77.842,172.270,29.741,155.490
C02478=1062.476,125.734,-77.862,172.272,29.744,155.491
C02479=1062.482,125.983,-77.882,172.274,29.746,155.491
C02480=1062.489,126.267,-77.905,172.275,29.749,155.492
C02481=1062.496,126.552,-77.928,172.278,29.753,155.492
C02482=1062.503,126.835,-77.951,172.280,29.755,155.493
C02483=1062.509,127.120,-77.975,172.281,29.759,155.493
C02484=1062.515,127.369,-77.995,172.283,29.761,155.494
C02485=1062.521,127.618,-78.015,172.285,29.764,155.494
C02486=1062.527,127.867,-78.035,172.287,29.767,155.494
C02487=1062.533,128.116,-78.055,172.288,29.769,155.495
C02488=1062.539,128.365,-78.075,172.290,29.772,155.495
C02489=1062.545,128.614,-78.095,172.292,29.775,155.496
C02490=1062.551,128.864,-78.116,172.293,29.778,155.496
C02491=1062.557,129.113,-78.136,172.295,29.780,155.496
C02492=1062.563,129.361,-78.156,172.297,29.782,155.497
C02493=1062.569,129.611,-78.177,172.299,29.785,155.497
C02494=1062.575,129.860,-78.197,172.300,29.788,155.497
C02495=1062.581,130.109,-78.217,172.302,29.791,155.498
C02496=1062.587,130.359,-78.238,172.304,29.793,155.498
C02497=1062.593,130.608,-78.258,172.305,29.796,155.499
C02498=1062.599,130.856,-78.279,172.307,29.799,155.499
C02499=1062.605,131.106,-78.300,172.309,29.801,155.500
C02500=1062.611,131.354,-78.320,172.311,29.804,155.500
C02501=1062.617,131.603,-78.339,172.311,29.807,155.500
C02502=1062.623,131.853,-78.360,172.313,29.809,155.501
C02503=1062.629,132.102,-78.380,172.315,29.812,155.501
C02504=1062.634,132.351,-78.401,172.316,29.815,155.502
C02505=1062.640,132.600,-78.423,172.318,29.817,155.502
C02506=1062.646,132.849,-78.443,172.320,29.820,155.502
C02507=1062.652,133.098,-78.463,172.322,29.823,155.503
C02508=1062.658,133.347,-78.483,172.323,29.825,155.503
C02509=1062.663,133.597,-78.504,172.325,29.828,155.504
C02510=1062.670,133.845,-78.525,172.327,29.831,155.504
C02511=1062.675,134.094,-78.545,172.328,29.834,155.505
C02512=1062.681,134.344,-78.566,172.330,29.837,155.505
C02513=1062.687,134.593,-78.586,172.332,29.840,155.505
C02514=1062.692,134.841,-78.607,172.334,29.842,155.506
C02515=1062.699,135.091,-78.628,172.335,29.845,155.506
C02516=1062.704,135.340,-78.648,172.337,29.848,155.507
C02517=1062.710,135.589,-78.670,172.339,29.850,155.507
C02518=1062.716,135.838,-78.690,172.340,29.853,155.507
C02519=1062.722,136.087,-78.710,172.342,29.856,155.508
C02520=1062.727,136.337,-78.731,172.344,29.858,155.508
C02521=1062.734,136.585,-78.752,172.346,29.861,155.509
C02522=1062.739,136.834,-78.772,172.347,29.864,155.509
C02523=1062.746,137.084,-78.793,172.349,29.866,155.509
C02524=1062.751,137.332,-78.814,172.351,29.869,155.510
C02525=1062.757,137.582,-78.835,172.352,29.872,155.510
C02526=1062.763,137.830,-78.856,172.354,29.875,155.511
C02527=1062.769,138.079,-78.876,172.356,29.877,155.511
C02528=1062.774,138.329,-78.897,172.358,29.880,155.512
C02529=1062.781,138.577,-78.918,172.359,29.883,155.512
C02530=1062.787,138.827,-78.939,172.361,29.886,155.512
C02531=1062.792,139.076,-78.960,172.363,29.889,155.513
C02532=1062.798,139.325,-78.981,172.364,29.891,155.513
C02533=1062.804,139.574,-79.001,172.366,29.894,155.514
C02534=1062.810,139.823,-79.022,172.368,29.897,155.514
C02535=1062.815,140.073,-79.043,172.370,29.899,155.514
C02536=1062.822,140.321,-79.064,172.371,29.902,155.515
C02537=1062.828,140.571,-79.085,172.373,29.905,155.515
C02538=1062.833,140.819,-79.106,172.375,29.908,155.516
C02539=1062.838,141.068,-79.127,172.376,29.910,155.516
C02540=1062.845,141.317,-79.148,172.378,29.913,155.517
C02541=1062.850,141.567,-79.169,172.380,29.916,155.517
C02542=1062.856,141.816,-79.190,172.381,29.919,155.517
C02543=1062.862,142.065,-79.210,172.383,29.922,155.518
C02544=1062.869,142.349,-79.234,172.386,29.924,155.518
C02545=1062.875,142.633,-79.259,172.388,29.928,155.519
C02546=1062.881,142.917,-79.283,172.389,29.931,155.519
C02547=1062.888,143.201,-79.307,172.392,29.934,155.520
C02548=1062.894,143.450,-79.329,172.394,29.937,155.520
C02549=1062.901,143.699,-79.349,172.395,29.940,155.521
C02550=1062.906,143.948,-79.370,172.397,29.943,155.521
C02551=1062.912,144.197,-79.391,172.399,29.945,155.521
C02552=1062.917,144.446,-79.412,172.400,29.948,155.522
C02553=1062.923,144.695,-79.434,172.402,29.951,155.522
C02554=1062.929,144.944,-79.455,172.404,29.953,155.523
C02555=1062.935,145.194,-79.476,172.406,29.956,155.523
C02556=1062.940,145.442,-79.497,172.407,29.959,155.524
C02557=1062.947,145.691,-79.518,172.409,29.961,155.524
C02558=1062.953,145.941,-79.539,172.411,29.964,155.524
C02559=1062.959,146.189,-79.560,172.413,29.967,155.525
C02560=1062.965,146.438,-79.582,172.414,29.970,155.525
C02561=1062.970,146.688,-79.602,172.416,29.973,155.526
C02562=1062.976,146.937,-79.624,172.418,29.975,155.526
C02563=1062.982,147.185,-79.645,172.419,29.978,155.527
C02564=1062.988,147.434,-79.667,172.421,29.981,155.527
C02565=1062.993,147.684,-79.688,172.423,29.983,155.527
C02566=1062.999,147.933,-79.709,172.425,29.986,155.528
C02567=1063.005,148.181,-79.730,172.426,29.989,155.528
C02568=1063.011,148.431,-79.752,172.429,29.992,155.529
C02569=1063.017,148.680,-79.774,172.431,29.995,155.529
C02570=1063.023,148.929,-79.794,172.432,29.998,155.529
C02571=1063.029,149.178,-79.816,172.434,30.000,155.530
C02572=1063.034,149.427,-79.837,172.436,30.003,155.530
C02573=1063.040,149.676,-79.859,172.438,30.006,155.531
C02574=1063.046,149.924,-79.880,172.439,30.008,155.531
C02575=1063.052,150.173,-79.902,172.441,30.011,155.532
C02576=1063.057,150.423,-79.922,172.443,30.014,155.532
C02577=1063.064,150.672,-79.944,172.444,30.017,155.532
C02578=1063.070,150.921,-79.966,172.446,30.020,155.533
C02579=1063.075,151.170,-79.987,172.448,30.022,155.533
C02580=1063.081,151.419,-80.009,172.450,30.025,155.534
C02581=1063.086,151.668,-80.030,172.451,30.028,155.534
C02582=1063.092,151.917,-80.052,172.453,30.031,155.535
C02583=1063.098,152.165,-80.073,172.456,30.034,155.535
C02584=1063.104,152.414,-80.095,172.457,30.037,155.535
C02585=1063.110,152.664,-80.116,172.459,30.039,155.536
C02586=1063.116,152.912,-80.138,172.461,30.042,155.536
C02587=1063.121,153.162,-80.160,172.463,30.045,155.537
C02588=1063.128,153.411,-80.182,172.464,30.048,155.537
C02589=1063.133,153.660,-80.202,172.466,30.051,155.538
C02590=1063.139,153.909,-80.224,172.468,30.053,155.538
C02591=1063.144,154.158,-80.245,172.470,30.056,155.538
C02592=1063.151,154.406,-80.267,172.471,30.059,155.539
C02593=1063.157,154.655,-80.289,172.473,30.061,155.539
C02594=1063.162,154.904,-80.311,172.476,30.064,155.540
C02595=1063.168,155.154,-80.333,172.477,30.067,155.540
C02596=1063.174,155.403,-80.354,172.479,30.070,155.541
C02597=1063.180,155.651,-80.375,172.481,30.073,155.541
C02598=1063.185,155.901,-80.398,172.483,30.075,155.541
C02599=1063.191,156.150,-80.419,172.484,30.078,155.542
C02600=1063.197,156.398,-80.441,172.486,30.081,155.542
C02601=1063.203,156.648,-80.462,172.488,30.084,155.543
C02602=1063.209,156.897,-80.484,172.490,30.087,155.543
C02603=1063.214,157.146,-80.506,172.492,30.090,155.544
C02604=1063.221,157.394,-80.528,172.494,30.092,155.544
C02605=1063.226,157.644,-80.550,172.496,30.095,155.545
C02606=1063.232,157.892,-80.572,172.497,30.098,155.545
C02607=1063.238,158.141,-80.593,172.499,30.101,155.545
C02608=1063.244,158.425,-80.619,172.501,30.104,155.546
C02609=1063.251,158.709,-80.643,172.503,30.108,155.546
C02610=1063.257,158.993,-80.668,172.505,30.110,155.547
C02611=1063.264,159.276,-80.693,172.508,30.114,155.547
C02612=1063.270,159.526,-80.714,172.510,30.116,155.548
C02613=1063.276,159.775,-80.737,172.511,30.119,155.548
C02614=1063.282,160.024,-80.759,172.513,30.122,155.549
C02615=1063.288,160.272,-80.780,172.515,30.125,155.549
C02616=1063.293,160.522,-80.802,172.517,30.128,155.550
C02617=1063.300,160.770,-80.825,172.519,30.130,155.550
C02618=1063.306,161.020,-80.846,172.521,30.133,155.550
C02619=1063.311,161.268,-80.868,172.523,30.136,155.551
C02620=1063.316,161.518,-80.890,172.524,30.139,155.551
C02621=1063.322,161.766,-80.913,172.526,30.142,155.552
C02622=1063.327,162.015,-80.935,172.528,30.145,155.552
C02623=1063.333,162.264,-80.958,172.530,30.148,155.553
C02624=1063.339,162.513,-80.979,172.531,30.151,155.553
C02625=1063.344,162.762,-81.001,172.534,30.154,155.554
C02626=1063.350,163.011,-81.024,172.536,30.156,155.554
C02627=1063.356,163.260,-81.046,172.537,30.160,155.554
C02628=1063.361,163.509,-81.067,172.539,30.162,155.555
C02629=1063.367,163.758,-81.090,172.541,30.165,155.555
C02630=1063.373,164.007,-81.112,172.543,30.168,155.556
C02631=1063.378,164.255,-81.135,172.544,30.171,155.556
C02632=1063.384,164.505,-81.156,172.547,30.174,155.557
C02633=1063.390,164.754,-81.179,172.549,30.177,155.557
C02634=1063.395,165.003,-81.201,172.550,30.180,155.558
C02635=1063.400,165.251,-81.224,172.552,30.183,155.558
C02636=1063.406,165.500,-81.246,172.554,30.186,155.559
C02637=1063.412,165.749,-81.269,172.556,30.188,155.559
C02638=1063.418,165.999,-81.291,172.558,30.192,155.559
C02639=1063.423,166.247,-81.313,172.560,30.194,155.560
C02640=1063.429,166.496,-81.335,172.562,30.198,155.560
C02641=1063.435,166.745,-81.358,172.564,30.200,155.561
C02642=1063.441,166.994,-81.380,172.565,30.203,155.561
C02643=1063.446,167.243,-81.402,172.567,30.206,155.562
C02644=1063.451,167.492,-81.424,172.570,30.209,155.562
C02645=1063.457,167.741,-81.447,172.571,30.212,155.563
C02646=1063.463,167.990,-81.469,172.573,30.215,155.563
C02647=1063.469,168.239,-81.492,172.575,30.218,155.564
C02648=1063.475,168.488,-81.515,172.577,30.220,155.564
C02649=1063.480,168.736,-81.536,172.578,30.223,155.564
C02650=1063.486,168.985,-81.559,172.581,30.226,155.565
C02651=1063.491,169.235,-81.581,172.583,30.229,155.565
C02652=1063.497,169.484,-81.604,172.585,30.232,155.566
C02653=1063.504,169.732,-81.627,172.586,30.235,155.566
C02654=1063.509,169.982,-81.649,172.588,30.238,155.567
C02655=1063.514,170.230,-81.671,172.591,30.241,155.567
C02656=1063.521,170.479,-81.694,172.592,30.244,155.568
C02657=1063.526,170.728,-81.716,172.594,30.247,155.568
C02658=1063.532,170.977,-81.739,172.596,30.250,155.569
C02659=1063.537,171.226,-81.762,172.598,30.252,155.569
C02660=1063.544,171.475,-81.784,172.600,30.256,155.569
C02661=1063.549,171.724,-81.807,172.602,30.258,155.570
C02662=1063.555,171.973,-81.829,172.604,30.261,155.570
C02663=1063.560,172.221,-81.852,172.606,30.264,155.571
C02664=1063.566,172.470,-81.875,172.607,30.267,155.571
C02665=1063.572,172.719,-81.897,172.610,30.270,155.572
C02666=1063.578,172.968,-81.920,172.612,30.273,155.572
C02667=1063.584,173.217,-81.943,172.613,30.276,155.573
C02668=1063.589,173.466,-81.965,172.615,30.278,155.573
C02669=1063.595,173.715,-81.987,172.618,30.282,155.573
C02670=1063.601,173.964,-82.010,172.620,30.284,155.574
C02671=1063.607,174.213,-82.033,172.621,30.287,155.574
C02672=1063.613,174.496,-82.059,172.624,30.290,155.575
C02673=1063.620,174.780,-82.084,172.626,30.294,155.575
C02674=1063.626,175.063,-82.110,172.628,30.297,155.576
C02675=1063.633,175.346,-82.136,172.630,30.300,155.576
C02676=1063.639,175.595,-82.159,172.633,30.303,155.577
C02677=1063.645,175.844,-82.182,172.635,30.306,155.577
C02678=1063.651,176.092,-82.205,172.636,30.309,155.578
C02679=1063.656,176.342,-82.227,172.638,30.312,155.578
C02680=1063.662,176.591,-82.250,172.641,30.315,155.579
C02681=1063.668,176.840,-82.273,172.643,30.318,155.579
C02682=1063.674,177.088,-82.295,172.644,30.320,155.579
C02683=1063.680,177.337,-82.318,172.646,30.324,155.580
C02684=1063.686,177.587,-82.341,172.649,30.326,155.580
C02685=1063.692,177.836,-82.364,172.651,30.329,155.581
C02686=1063.698,178.085,-82.387,172.652,30.332,155.581
C02687=1063.703,178.334,-82.410,172.654,30.335,155.582
C02688=1063.710,178.582,-82.433,172.657,30.338,155.582
C02689=1063.716,178.831,-82.456,172.658,30.341,155.583
C02690=1063.721,179.080,-82.478,172.660,30.344,155.583
C02691=1063.727,179.329,-82.501,172.662,30.346,155.584
C02692=1063.733,179.578,-82.524,172.665,30.350,155.584
C02693=1063.739,179.827,-82.547,172.666,30.352,155.584
C02694=1063.745,180.075,-82.570,172.668,30.355,155.585
C02695=1063.751,180.324,-82.593,172.671,30.359,155.585
C02696=1063.757,180.573,-82.616,172.673,30.361,155.586
C02697=1063.763,180.821,-82.639,172.674,30.364,155.586
C02698=1063.769,181.071,-82.663,172.677,30.367,155.587
C02699=1063.775,181.320,-82.685,172.679,30.370,155.587
C02700=1063.780,181.569,-82.708,172.681,30.373,155.588
C02701=1063.786,181.818,-82.731,172.682,30.376,155.588
C02702=1063.793,182.066,-82.754,172.685,30.379,155.589
C02703=1063.798,182.315,-82.777,172.687,30.381,155.589
C02704=1063.804,182.563,-82.800,172.688,30.384,155.589
C02705=1063.811,182.813,-82.824,172.691,30.387,155.590
C02706=1063.816,183.062,-82.847,172.693,30.390,155.590
C02707=1063.822,183.311,-82.870,172.695,30.393,155.591
C02708=1063.828,183.560,-82.892,172.697,30.396,155.591
C02709=1063.834,183.808,-82.915,172.699,30.399,155.592
C02710=1063.840,184.056,-82.938,172.701,30.402,155.592
C02711=1063.847,184.306,-82.962,172.704,30.405,155.593
C02712=1063.852,184.555,-82.985,172.705,30.407,155.593
C02713=1063.857,184.804,-83.008,172.707,30.411,155.594
C02714=1063.863,185.052,-83.032,172.710,30.414,155.594
C02715=1063.869,185.301,-83.055,172.712,30.417,155.594
C02716=1063.874,185.551,-83.078,172.713,30.420,155.595
C02717=1063.880,185.799,-83.102,172.715,30.423,155.596
C02718=1063.886,186.048,-83.125,172.718,30.426,155.596
C02719=1063.891,186.297,-83.149,172.720,30.429,155.596
C02720=1063.897,186.545,-83.172,172.721,30.432,155.597
C02721=1063.903,186.794,-83.195,172.724,30.435,155.597
C02722=1063.909,187.043,-83.220,172.726,30.438,155.598
C02723=1063.914,187.292,-83.243,172.727,30.441,155.598
C02724=1063.920,187.541,-83.266,172.730,30.444,155.599
C02725=1063.925,187.790,-83.290,172.732,30.448,155.599
C02726=1063.931,188.039,-83.313,172.734,30.450,155.600
C02727=1063.936,188.287,-83.337,172.736,30.454,155.600
C02728=1063.942,188.536,-83.360,172.738,30.456,155.601
C02729=1063.948,188.784,-83.384,172.740,30.460,155.601
C02730=1063.954,189.034,-83.408,172.743,30.463,155.602
C02731=1063.960,189.283,-83.431,172.744,30.466,155.602
C02732=1063.966,189.531,-83.454,172.746,30.469,155.603
C02733=1063.971,189.780,-83.479,172.749,30.472,155.603
C02734=1063.977,190.029,-83.501,172.751,30.475,155.604
C02735=1063.982,190.278,-83.526,172.752,30.478,155.604
C02736=1063.989,190.561,-83.552,172.755,30.481,155.605
C02737=1063.995,190.844,-83.579,172.758,30.485,155.605
C02738=1064.002,191.127,-83.606,172.760,30.489,155.606
C02739=1064.008,191.410,-83.633,172.762,30.492,155.606
C02740=1064.014,191.658,-83.656,172.765,30.495,155.607
C02741=1064.020,191.908,-83.681,172.767,30.498,155.607
C02742=1064.026,192.157,-83.704,172.768,30.501,155.608
C02743=1064.031,192.405,-83.728,172.771,30.504,155.608
C02744=1064.037,192.653,-83.752,172.773,30.507,155.609
C02745=1064.043,192.903,-83.775,172.774,30.510,155.609
C02746=1064.049,193.152,-83.800,172.777,30.513,155.610
C02747=1064.055,193.400,-83.823,172.779,30.516,155.610
C02748=1064.060,193.649,-83.847,172.782,30.520,155.611
C02749=1064.066,193.898,-83.871,172.783,30.523,155.611
C02750=1064.072,194.147,-83.895,172.785,30.526,155.612
C02751=1064.077,194.396,-83.918,172.788,30.529,155.612
C02752=1064.084,194.645,-83.942,172.790,30.532,155.613
C02753=1064.089,194.893,-83.966,172.792,30.535,155.613
C02754=1064.095,195.142,-83.989,172.794,30.538,155.614
C02755=1064.100,195.391,-84.013,172.796,30.541,155.614
C02756=1064.107,195.640,-84.037,172.799,30.544,155.615
C02757=1064.112,195.888,-84.062,172.800,30.547,155.615
C02758=1064.118,196.136,-84.085,172.803,30.550,155.616
C02759=1064.124,196.386,-84.109,172.805,30.554,155.616
C02760=1064.130,196.635,-84.133,172.807,30.556,155.617
C02761=1064.135,196.883,-84.157,172.809,30.560,155.617
C02762=1064.142,197.132,-84.181,172.811,30.563,155.618
C02763=1064.147,197.381,-84.206,172.814,30.566,155.618
C02764=1064.153,197.630,-84.229,172.816,30.569,155.619
C02765=1064.159,197.879,-84.253,172.818,30.572,155.619
C02766=1064.165,198.127,-84.277,172.820,30.575,155.620
C02767=1064.171,198.377,-84.301,172.822,30.578,155.620
C02768=1064.177,198.625,-84.325,172.824,30.581,155.621
C02769=1064.182,198.873,-84.349,172.826,30.584,155.621
C02770=1064.189,199.122,-84.373,172.829,30.587,155.622
C02771=1064.194,199.371,-84.398,172.831,30.591,155.622
C02772=1064.201,199.620,-84.422,172.833,30.593,155.622
C02773=1064.206,199.869,-84.446,172.835,30.597,155.623
C02774=1064.213,200.118,-84.470,172.838,30.600,155.624
C02775=1064.218,200.366,-84.494,172.840,30.603,155.624
C02776=1064.224,200.614,-84.518,172.842,30.606,155.624
C02777=1064.230,200.864,-84.542,172.844,30.609,155.625
C02778=1064.236,201.112,-84.566,172.846,30.612,155.625
C02779=1064.242,201.361,-84.591,172.849,30.615,155.626
C02780=1064.248,201.609,-84.614,172.850,30.618,155.626
C02781=1064.254,201.859,-84.639,172.853,30.621,155.627
C02782=1064.260,202.107,-84.663,172.855,30.624,155.627
C02783=1064.266,202.356,-84.687,172.858,30.628,155.628
C02784=1064.271,202.605,-84.712,172.859,30.631,155.628
C02785=1064.276,202.854,-84.736,172.862,30.634,155.629
C02786=1064.282,203.103,-84.760,172.864,30.637,155.629
C02787=1064.288,203.351,-84.784,172.867,30.640,155.630
C02788=1064.294,203.600,-84.809,172.868,30.644,155.630
C02789=1064.299,203.849,-84.833,172.871,30.647,155.631
C02790=1064.306,204.098,-84.858,172.873,30.650,155.632
C02791=1064.311,204.346,-84.883,172.876,30.653,155.632
C02792=1064.317,204.595,-84.907,172.877,30.657,155.633
C02793=1064.323,204.844,-84.931,172.880,30.659,155.633
C02794=1064.328,205.092,-84.955,172.882,30.663,155.634
C02795=1064.334,205.341,-84.980,172.885,30.666,155.634
C02796=1064.340,205.590,-85.005,172.886,30.669,155.635
C02797=1064.345,205.839,-85.029,172.889,30.673,155.635
C02798=1064.351,206.087,-85.053,172.891,30.676,155.636
C02799=1064.358,206.336,-85.078,172.893,30.679,155.636
C02800=1064.382,207.383,-85.181,173.055,30.759,155.642
C02801=1064.387,207.605,-85.204,173.057,30.762,155.643
C02802=1064.393,207.827,-85.226,173.059,30.766,155.644
C02803=1064.398,208.050,-85.249,173.061,30.769,155.644
C02804=1064.404,208.272,-85.273,173.062,30.773,155.645
C02805=1064.409,208.494,-85.294,173.064,30.777,155.646
C02806=1064.414,208.716,-85.318,173.066,30.781,155.646
C02807=1064.420,208.939,-85.340,173.067,30.784,155.647
C02808=1064.425,209.162,-85.363,173.069,30.787,155.647
C02809=1064.431,209.411,-85.388,173.071,30.792,155.648
C02810=1064.437,209.659,-85.414,173.074,30.796,155.649
C02811=1064.443,209.907,-85.439,173.075,30.800,155.650
C02812=1064.449,210.155,-85.465,173.077,30.804,155.650
C02813=1064.455,210.404,-85.491,173.079,30.808,155.651
C02814=1064.461,210.653,-85.516,173.081,30.812,155.652
C02815=1064.467,210.902,-85.541,173.083,30.816,155.653
C02816=1064.473,211.150,-85.567,173.085,30.821,155.653
C02817=1064.479,211.399,-85.593,173.087,30.824,155.654
C02818=1064.485,211.648,-85.618,173.089,30.829,155.655
C02819=1064.491,211.897,-85.643,173.091,30.832,155.655
C02820=1064.498,212.145,-85.669,173.093,30.837,155.656
C02821=1064.503,212.394,-85.695,173.095,30.841,155.657
C02822=1064.509,212.642,-85.721,173.097,30.845,155.658
C02823=1064.516,212.891,-85.746,173.099,30.849,155.658
C02824=1064.521,213.140,-85.772,173.101,30.853,155.659
C02825=1064.527,213.389,-85.797,173.103,30.857,155.660
C02826=1064.533,213.637,-85.824,173.105,30.861,155.661
C02827=1064.539,213.885,-85.849,173.107,30.865,155.661
C02828=1064.545,214.134,-85.874,173.109,30.869,155.662
C02829=1064.550,214.383,-85.900,173.111,30.874,155.663
C02830=1064.557,214.631,-85.926,173.113,30.877,155.663
C02831=1064.562,214.880,-85.952,173.115,30.882,155.664
C02832=1064.569,215.128,-85.977,173.117,30.886,155.665
C02833=1064.574,215.377,-86.004,173.119,30.890,155.666
C02834=1064.581,215.625,-86.029,173.121,30.894,155.666
C02835=1064.587,215.874,-86.055,173.123,30.898,155.667
C02836=1064.593,216.122,-86.081,173.125,30.902,155.668
C02837=1064.599,216.371,-86.107,173.127,30.906,155.669
C02838=1064.604,216.620,-86.133,173.130,30.910,155.669
C02839=1064.611,216.868,-86.159,173.131,30.914,155.670
C02840=1064.616,217.117,-86.185,173.133,30.918,155.671
C02841=1064.623,217.365,-86.211,173.136,30.922,155.671
C02842=1064.628,217.614,-86.237,173.137,30.926,155.672
C02843=1064.635,217.863,-86.262,173.139,30.930,155.673
C02844=1064.641,218.112,-86.289,173.141,30.934,155.673
C02845=1064.647,218.360,-86.314,173.144,30.938,155.674
C02846=1064.653,218.609,-86.341,173.145,30.942,155.675
C02847=1064.659,218.857,-86.366,173.147,30.946,155.676
C02848=1064.665,219.106,-86.393,173.150,30.951,155.676
C02849=1064.671,219.354,-86.418,173.152,30.954,155.677
C02850=1064.677,219.603,-86.445,173.153,30.959,155.678
C02851=1064.683,219.851,-86.470,173.156,30.962,155.678
C02852=1064.689,220.100,-86.497,173.158,30.966,155.679
C02853=1064.695,220.349,-86.522,173.160,30.971,155.680
C02854=1064.701,220.598,-86.549,173.162,30.974,155.681
C02855=1064.707,220.846,-86.575,173.164,30.979,155.681
C02856=1064.713,221.095,-86.601,173.167,30.983,155.682
C02857=1064.719,221.319,-86.625,173.168,30.986,155.683
C02858=1064.724,221.544,-86.648,173.170,30.990,155.683
C02859=1064.729,221.768,-86.672,173.172,30.994,155.684
C02860=1064.735,221.993,-86.695,173.174,30.997,155.685
C02861=1064.740,222.218,-86.719,173.175,31.001,155.685
C02862=1064.746,222.442,-86.743,173.177,31.004,155.686
C02863=1064.751,222.668,-86.767,173.179,31.008,155.687
C02864=1064.757,222.892,-86.791,173.182,31.012,155.687
C02865=1064.763,223.141,-86.817,173.183,31.016,155.688
C02866=1064.768,223.389,-86.844,173.185,31.020,155.689
C02867=1064.775,223.638,-86.869,173.188,31.024,155.689
C02868=1064.780,223.886,-86.896,173.190,31.028,155.690
C02869=1064.786,224.134,-86.923,173.191,31.032,155.691
C02870=1064.793,224.383,-86.950,173.194,31.036,155.692
C02871=1064.799,224.632,-86.975,173.196,31.040,155.692
C02872=1064.805,224.880,-87.002,173.198,31.044,155.693
C02873=1064.810,225.129,-87.028,173.200,31.048,155.694
C02874=1064.816,225.377,-87.055,173.202,31.052,155.694
C02875=1064.822,225.626,-87.080,173.205,31.056,155.695
C02876=1064.829,225.875,-87.107,173.207,31.060,155.696
C02877=1064.834,226.123,-87.134,173.208,31.064,155.697
C02878=1064.840,226.372,-87.160,173.211,31.068,155.697
C02879=1064.846,226.620,-87.187,173.213,31.072,155.698
C02880=1064.853,226.869,-87.214,173.215,31.076,155.699
C02881=1064.859,227.117,-87.240,173.217,31.080,155.699
C02882=1064.864,227.366,-87.266,173.219,31.084,155.700
C02883=1064.870,227.614,-87.293,173.222,31.088,155.701
C02884=1064.876,227.863,-87.320,173.224,31.092,155.701
C02885=1064.883,228.111,-87.346,173.226,31.096,155.702
C02886=1064.889,228.360,-87.373,173.228,31.100,155.703
C02887=1064.895,228.608,-87.399,173.230,31.104,155.704
C02888=1064.901,228.857,-87.426,173.232,31.108,155.704
C02889=1064.907,229.106,-87.453,173.234,31.112,155.705
C02890=1064.913,229.354,-87.479,173.237,31.116,155.706
C02891=1064.920,229.603,-87.506,173.239,31.120,155.706
C02892=1064.925,229.851,-87.533,173.241,31.124,155.707
C02893=1064.931,230.099,-87.559,173.243,31.128,155.708
C02894=1064.937,230.348,-87.586,173.245,31.132,155.709
C02895=1064.943,230.597,-87.613,173.248,31.136,155.709
C02896=1064.949,230.845,-87.639,173.249,31.140,155.710
C02897=1064.955,231.094,-87.666,173.252,31.144,155.711
C02898=1064.961,231.343,-87.693,173.254,31.148,155.711
C02899=1064.967,231.590,-87.721,173.256,31.152,155.712
C02900=1064.973,231.839,-87.747,173.259,31.156,155.713
C02901=1064.979,232.087,-87.774,173.260,31.160,155.714
C02902=1064.985,232.336,-87.801,173.263,31.164,155.714
C02903=1064.991,232.585,-87.827,173.265,31.168,155.715
C02904=1064.997,232.833,-87.854,173.268,31.172,155.716
C02905=1065.003,233.082,-87.881,173.269,31.176,155.716
C02906=1065.009,233.330,-87.909,173.272,31.180,155.717
C02907=1065.016,233.579,-87.936,173.274,31.184,155.718
C02908=1065.021,233.827,-87.963,173.276,31.188,155.719
C02909=1065.026,234.076,-87.989,173.278,31.192,155.719
C02910=1065.032,234.323,-88.017,173.280,31.195,155.720
C02911=1065.039,234.573,-88.044,173.283,31.200,155.721
C02912=1065.045,234.821,-88.070,173.285,31.204,155.721
C02913=1065.050,235.041,-88.095,173.286,31.207,155.722
C02914=1065.055,235.262,-88.119,173.289,31.211,155.723
C02915=1065.061,235.483,-88.142,173.291,31.214,155.723
C02916=1065.067,235.704,-88.167,173.293,31.218,155.724
C02917=1065.071,235.925,-88.191,173.295,31.222,155.725
C02918=1065.076,236.146,-88.215,173.296,31.225,155.725
C02919=1065.082,236.366,-88.240,173.299,31.229,155.726
C02920=1065.087,236.587,-88.263,173.301,31.232,155.726
C02921=1065.093,236.835,-88.291,173.303,31.236,155.727
C02922=1065.099,237.084,-88.318,173.305,31.240,155.728
C02923=1065.105,237.332,-88.344,173.307,31.244,155.729
C02924=1065.112,237.580,-88.372,173.310,31.248,155.729
C02925=1065.117,237.829,-88.399,173.312,31.252,155.730
C02926=1065.123,238.077,-88.427,173.314,31.256,155.731
C02927=1065.129,238.326,-88.454,173.316,31.260,155.731
C02928=1065.135,238.574,-88.481,173.319,31.264,155.732
C02929=1065.142,238.823,-88.508,173.321,31.268,155.733
C02930=1065.147,239.071,-88.536,173.324,31.272,155.733
C02931=1065.154,239.320,-88.563,173.325,31.276,155.734
C02932=1065.160,239.568,-88.590,173.328,31.280,155.735
C02933=1065.166,239.817,-88.617,173.330,31.284,155.736
C02934=1065.171,240.065,-88.645,173.333,31.288,155.736
C02935=1065.178,240.314,-88.672,173.334,31.292,155.737
C02936=1065.184,240.561,-88.700,173.337,31.296,155.738
C02937=1065.190,240.810,-88.727,173.339,31.300,155.738
C02938=1065.196,241.059,-88.755,173.342,31.304,155.739
C02939=1065.202,241.307,-88.783,173.344,31.307,155.740
C02940=1065.208,241.555,-88.809,173.346,31.312,155.741
C02941=1065.214,241.804,-88.837,173.348,31.315,155.741
C02942=1065.220,242.052,-88.864,173.351,31.319,155.742
C02943=1065.226,242.301,-88.892,173.353,31.323,155.743
C02944=1065.232,242.549,-88.920,173.355,31.327,155.743
C02945=1065.238,242.798,-88.947,173.357,31.331,155.744
C02946=1065.243,243.046,-88.975,173.360,31.335,155.745
C02947=1065.250,243.295,-89.003,173.362,31.339,155.745
C02948=1065.255,243.543,-89.030,173.365,31.343,155.746
C02949=1065.262,243.792,-89.057,173.366,31.347,155.747
C02950=1065.267,244.040,-89.085,173.369,31.351,155.748
C02951=1065.274,244.288,-89.113,173.372,31.355,155.748
C02952=1065.280,244.537,-89.142,173.374,31.359,155.749
C02953=1065.286,244.785,-89.169,173.376,31.363,155.750
C02954=1065.292,245.034,-89.196,173.378,31.367,155.750
C02955=1065.298,245.282,-89.224,173.381,31.371,155.751
C02956=1065.304,245.530,-89.252,173.383,31.375,155.752
C02957=1065.310,245.778,-89.280,173.386,31.379,155.753
C02958=1065.316,246.027,-89.308,173.387,31.383,155.753
C02959=1065.322,246.275,-89.335,173.390,31.387,155.754
C02960=1065.328,246.523,-89.364,173.392,31.391,155.755
C02961=1065.334,246.773,-89.391,173.395,31.395,155.755
C02962=1065.339,247.021,-89.419,173.397,31.399,155.756
C02963=1065.345,247.269,-89.447,173.399,31.403,155.757
C02964=1065.351,247.517,-89.474,173.402,31.407,155.758
C02965=1065.357,247.766,-89.503,173.404,31.411,155.758
C02966=1065.363,248.014,-89.530,173.407,31.415,155.759
C02967=1065.369,248.263,-89.559,173.408,31.419,155.760
C02968=1065.375,248.511,-89.587,173.411,31.423,155.761
C02969=1065.380,248.729,-89.612,173.413,31.426,155.761
C02970=1065.385,248.945,-89.636,173.415,31.430,155.762
C02971=1065.390,249.163,-89.660,173.418,31.434,155.762
C02972=1065.396,249.380,-89.685,173.419,31.437,155.763
C02973=1065.400,249.598,-89.710,173.421,31.441,155.764
C02974=1065.406,249.816,-89.734,173.423,31.444,155.764
C02975=1065.411,250.033,-89.759,173.426,31.448,155.765
C02976=1065.416,250.251,-89.783,173.428,31.451,155.766
C02977=1065.422,250.499,-89.812,173.430,31.455,155.766
C02978=1065.428,250.747,-89.840,173.432,31.459,155.767
C02979=1065.434,250.996,-89.868,173.435,31.463,155.768
C02980=1065.440,251.245,-89.896,173.437,31.467,155.768
C02981=1065.446,251.492,-89.925,173.440,31.471,155.769
C02982=1065.452,251.741,-89.953,173.442,31.475,155.770
C02983=1065.458,251.990,-89.981,173.444,31.479,155.771
C02984=1065.464,252.237,-90.009,173.447,31.483,155.771
C02985=1065.470,252.486,-90.037,173.449,31.487,155.772
C02986=1065.476,252.734,-90.066,173.452,31.491,155.773
C02987=1065.482,252.983,-90.094,173.454,31.495,155.773
C02988=1065.487,253.231,-90.122,173.456,31.499,155.774
C02989=1065.494,253.479,-90.150,173.459,31.503,155.775
C02990=1065.500,253.728,-90.179,173.461,31.507,155.775
C02991=1065.506,253.976,-90.207,173.464,31.511,155.776
C02992=1065.512,254.224,-90.235,173.466,31.515,155.777
C02993=1065.518,254.473,-90.264,173.468,31.519,155.778
C02994=1065.524,254.721,-90.293,173.471,31.523,155.778
C02995=1065.530,254.969,-90.320,173.474,31.527,155.779
C02996=1065.536,255.217,-90.349,173.476,31.530,155.780
C02997=1065.542,255.466,-90.377,173.478,31.535,155.780
C02998=1065.548,255.715,-90.406,173.480,31.538,155.781
C02999=1065.554,255.963,-90.435,173.483,31.542,155.782
C03000=1065.560,256.211,-90.463,173.486,31.547,155.783
C03001=1065.567,256.459,-90.491,173.488,31.550,155.783
C03002=1065.573,256.707,-90.519,173.490,31.555,155.784
C03003=1065.578,256.956,-90.548,173.493,31.558,155.785
C03004=1065.585,257.204,-90.577,173.495,31.562,155.785
C03005=1065.590,257.452,-90.605,173.498,31.566,155.786
C03006=1065.596,257.700,-90.634,173.501,31.570,155.787
C03007=1065.602,257.949,-90.662,173.503,31.574,155.788
C03008=1065.609,258.197,-90.691,173.505,31.578,155.788
C03009=1065.615,258.446,-90.719,173.508,31.582,155.789
C03010=1065.621,258.694,-90.748,173.510,31.586,155.790
C03011=1065.627,258.943,-90.776,173.513,31.590,155.790
C03012=1065.634,259.191,-90.805,173.516,31.594,155.791
C03013=1065.639,259.438,-90.834,173.517,31.598,155.792
C03014=1065.645,259.687,-90.862,173.520,31.601,155.792
C03015=1065.651,259.935,-90.891,173.523,31.606,155.793
C03016=1065.657,260.184,-90.920,173.526,31.610,155.794
C03017=1065.664,260.432,-90.948,173.528,31.613,155.795
C03018=1065.671,260.680,-90.977,173.530,31.617,155.795
C03019=1065.677,260.929,-91.005,173.533,31.621,155.796
C03020=1065.683,261.177,-91.034,173.535,31.625,155.797
C03021=1065.689,261.425,-91.064,173.538,31.629,155.797
C03022=1065.695,261.674,-91.092,173.541,31.633,155.798
C03023=1065.701,261.922,-91.121,173.543,31.637,155.799
C03024=1065.708,262.170,-91.150,173.545,31.641,155.800
C03025=1065.713,262.386,-91.175,173.548,31.644,155.800
C03026=1065.719,262.603,-91.199,173.550,31.648,155.801
C03027=1065.723,262.819,-91.225,173.552,31.651,155.801
C03028=1065.729,263.036,-91.250,173.555,31.654,155.802
C03029=1065.735,263.252,-91.275,173.557,31.658,155.803
C03030=1065.740,263.468,-91.301,173.558,31.661,155.803
C03031=1065.745,263.684,-91.326,173.561,31.664,155.804
C03032=1065.751,263.901,-91.351,173.563,31.668,155.804
C03033=1065.756,264.149,-91.380,173.566,31.672,155.805
C03034=1065.762,264.397,-91.409,173.569,31.676,155.806
C03035=1065.768,264.646,-91.438,173.571,31.680,155.807
C03036=1065.774,264.894,-91.467,173.573,31.684,155.807
C03037=1065.780,265.142,-91.496,173.576,31.688,155.808
C03038=1065.786,265.390,-91.525,173.578,31.692,155.809
C03039=1065.793,265.638,-91.554,173.581,31.696,155.809
C03040=1065.799,265.887,-91.583,173.584,31.700,155.810
C03041=1065.804,266.135,-91.613,173.587,31.704,155.811
C03042=1065.811,266.383,-91.642,173.588,31.708,155.812
C03043=1065.817,266.631,-91.671,173.591,31.712,155.812
C03044=1065.823,266.879,-91.700,173.594,31.716,155.813
C03045=1065.829,267.128,-91.730,173.597,31.720,155.814
C03046=1065.835,267.376,-91.759,173.599,31.724,155.815
C03047=1065.841,267.624,-91.788,173.601,31.728,155.815
C03048=1065.847,267.873,-91.818,173.604,31.732,155.816
C03049=1065.853,268.121,-91.847,173.607,31.736,155.817
C03050=1065.859,268.369,-91.876,173.609,31.740,155.817
C03051=1065.865,268.617,-91.905,173.612,31.744,155.818
C03052=1065.872,268.865,-91.935,173.615,31.748,155.819
C03053=1065.878,269.114,-91.964,173.617,31.752,155.820
C03054=1065.883,269.362,-91.994,173.619,31.756,155.820
C03055=1065.890,269.610,-92.023,173.622,31.760,155.821
C03056=1065.896,269.858,-92.052,173.625,31.764,155.822
C03057=1065.901,270.107,-92.082,173.628,31.768,155.823
C03058=1065.908,270.354,-92.112,173.630,31.772,155.823
C03059=1065.914,270.603,-92.141,173.632,31.775,155.824
C03060=1065.920,270.851,-92.170,173.635,31.780,155.825
C03061=1065.926,271.099,-92.199,173.638,31.784,155.825
C03062=1065.932,271.347,-92.230,173.641,31.788,155.826
C03063=1065.938,271.595,-92.259,173.643,31.792,155.827
C03064=1065.944,271.843,-92.288,173.646,31.796,155.828
C03065=1065.950,272.092,-92.318,173.648,31.800,155.828
C03066=1065.956,272.340,-92.348,173.651,31.804,155.829
C03067=1065.963,272.588,-92.377,173.654,31.808,155.830
C03068=1065.968,272.836,-92.407,173.656,31.812,155.831
C03069=1065.975,273.084,-92.436,173.659,31.816,155.831
C03070=1065.980,273.333,-92.466,173.662,31.820,155.832
C03071=1065.987,273.580,-92.496,173.664,31.824,155.833
C03072=1065.993,273.829,-92.526,173.667,31.828,155.833
C03073=1065.999,274.077,-92.556,173.669,31.832,155.834
C03074=1066.005,274.325,-92.585,173.672,31.836,155.835
C03075=1066.010,274.574,-92.615,173.675,31.840,155.836
C03076=1066.017,274.821,-92.645,173.678,31.844,155.836
C03077=1066.022,275.070,-92.674,173.681,31.848,155.837
C03078=1066.029,275.317,-92.704,173.682,31.852,155.838
C03079=1066.035,275.566,-92.734,173.685,31.856,155.839
C03080=1066.041,275.814,-92.764,173.688,31.860,155.839
C03081=1066.046,276.032,-92.790,173.691,31.863,155.840
C03082=1066.052,276.250,-92.817,173.693,31.867,155.841
C03083=1066.057,276.468,-92.843,173.696,31.871,155.841
C03084=1066.062,276.686,-92.869,173.698,31.874,155.842
C03085=1066.067,276.904,-92.896,173.700,31.878,155.842
C03086=1066.073,277.123,-92.922,173.702,31.881,155.843
C03087=1066.078,277.341,-92.949,173.705,31.885,155.844
C03088=1066.084,277.559,-92.975,173.707,31.888,155.844
C03089=1066.090,277.807,-93.004,173.710,31.892,155.845
C03090=1066.096,278.055,-93.035,173.713,31.897,155.846
C03091=1066.102,278.304,-93.065,173.716,31.901,155.847
C03092=1066.108,278.552,-93.095,173.717,31.905,155.847
C03093=1066.114,278.800,-93.125,173.720,31.909,155.848
C03094=1066.120,279.047,-93.155,173.723,31.913,155.849
C03095=1066.127,279.296,-93.185,173.726,31.917,155.850
C03096=1066.133,279.544,-93.215,173.729,31.921,155.850
C03097=1066.138,279.792,-93.245,173.732,31.925,155.851
C03098=1066.145,280.040,-93.276,173.734,31.929,155.852
C03099=1066.151,280.289,-93.305,173.737,31.933,155.853
C03100=1066.157,280.536,-93.335,173.739,31.937,155.853
C03101=1066.163,280.784,-93.366,173.742,31.941,155.854
C03102=1066.169,281.033,-93.397,173.745,31.945,155.855
C03103=1066.175,281.281,-93.427,173.748,31.949,155.856
C03104=1066.181,281.528,-93.457,173.751,31.953,155.856
C03105=1066.187,281.777,-93.488,173.753,31.957,155.857
C03106=1066.193,282.025,-93.518,173.756,31.962,155.858
C03107=1066.198,282.273,-93.548,173.759,31.965,155.859
C03108=1066.204,282.521,-93.578,173.761,31.970,155.859
C03109=1066.211,282.769,-93.608,173.764,31.974,155.860
C03110=1066.217,283.017,-93.639,173.767,31.978,155.861
C03111=1066.223,283.265,-93.669,173.770,31.982,155.862
C03112=1066.230,283.513,-93.700,173.772,31.986,155.862
C03113=1066.235,283.761,-93.730,173.775,31.990,155.863
C03114=1066.241,284.009,-93.761,173.778,31.994,155.864
C03115=1066.248,284.258,-93.791,173.781,31.998,155.865
C03116=1066.253,284.505,-93.822,173.784,32.002,155.865
C03117=1066.260,284.754,-93.852,173.787,32.007,155.866
C03118=1066.266,285.001,-93.883,173.789,32.010,155.867
C03119=1066.272,285.249,-93.914,173.792,32.015,155.868
C03120=1066.278,285.497,-93.944,173.794,32.018,155.868
C03121=1066.284,285.745,-93.975,173.797,32.023,155.869
C03122=1066.290,285.994,-94.005,173.800,32.027,155.870
C03123=1066.296,286.242,-94.036,173.803,32.031,155.871
C03124=1066.302,286.489,-94.066,173.806,32.035,155.871
C03125=1066.309,286.737,-94.098,173.809,32.039,155.872
C03126=1066.315,286.985,-94.128,173.812,32.043,155.873
C03127=1066.321,287.234,-94.159,173.814,32.047,155.874
C03128=1066.327,287.481,-94.189,173.817,32.051,155.874
C03129=1066.333,287.730,-94.220,173.820,32.055,155.875
C03130=1066.339,287.977,-94.251,173.823,32.060,155.876
C03131=1066.346,288.226,-94.282,173.826,32.063,155.877
C03132=1066.352,288.474,-94.312,173.829,32.068,155.877
C03133=1066.358,288.721,-94.343,173.832,32.072,155.878
C03134=1066.364,288.969,-94.374,173.834,32.076,155.879
C03135=1066.371,289.218,-94.404,173.836,32.080,155.880
C03136=1066.377,289.465,-94.435,173.839,32.084,155.880
C03137=1066.382,289.689,-94.464,173.842,32.088,155.881
C03138=1066.387,289.913,-94.491,173.845,32.092,155.882
C03139=1066.393,290.136,-94.519,173.847,32.095,155.882
C03140=1066.398,290.359,-94.547,173.850,32.099,155.883
C03141=1066.404,290.583,-94.575,173.853,32.103,155.884
C03142=1066.409,290.806,-94.603,173.855,32.106,155.885
C03143=1066.415,291.029,-94.631,173.857,32.110,155.885
C03144=1066.420,291.253,-94.658,173.860,32.114,155.886
C03145=1066.427,291.501,-94.690,173.863,32.118,155.887
C03146=1066.432,291.748,-94.720,173.866,32.122,155.887
C03147=1066.438,291.997,-94.752,173.869,32.127,155.888
C03148=1066.445,292.245,-94.783,173.872,32.130,155.889
C03149=1066.451,292.492,-94.814,173.875,32.135,155.890
C03150=1066.457,292.741,-94.845,173.878,32.139,155.891
C03151=1066.463,292.988,-94.876,173.880,32.143,155.891
C03152=1066.470,293.236,-94.908,173.883,32.148,155.892
C03153=1066.475,293.484,-94.938,173.886,32.151,155.893
C03154=1066.481,293.732,-94.970,173.889,32.156,155.894
C03155=1066.487,293.980,-95.000,173.892,32.160,155.894
C03156=1066.494,294.228,-95.032,173.895,32.164,155.895
C03157=1066.500,294.476,-95.064,173.898,32.168,155.896
C03158=1066.506,294.724,-95.094,173.901,32.172,155.897
C03159=1066.512,294.972,-95.126,173.904,32.176,155.897
C03160=1066.518,295.220,-95.158,173.906,32.181,155.898
C03161=1066.525,295.467,-95.189,173.909,32.185,155.899
C03162=1066.531,295.716,-95.219,173.912,32.189,155.900
C03163=1066.536,295.963,-95.251,173.915,32.193,155.901
C03164=1066.543,296.211,-95.283,173.918,32.197,155.901
C03165=1066.549,296.459,-95.315,173.921,32.201,155.902
C03166=1066.555,296.707,-95.346,173.924,32.206,155.903
C03167=1066.562,296.955,-95.376,173.927,32.210,155.904
C03168=1066.568,297.203,-95.408,173.930,32.214,155.905
C03169=1066.573,297.451,-95.440,173.932,32.219,155.905
C03170=1066.580,297.699,-95.472,173.935,32.223,155.906
C03171=1066.585,297.946,-95.503,173.938,32.227,155.907
C03172=1066.591,298.195,-95.535,173.941,32.231,155.908
C03173=1066.598,298.442,-95.567,173.944,32.236,155.909
C03174=1066.603,298.690,-95.598,173.947,32.240,155.909
C03175=1066.609,298.938,-95.630,173.950,32.244,155.910
C03176=1066.616,299.186,-95.662,173.954,32.249,155.911
C03177=1066.621,299.434,-95.693,173.957,32.253,155.912
C03178=1066.627,299.682,-95.725,173.959,32.257,155.913
C03179=1066.634,299.930,-95.757,173.962,32.261,155.913
C03180=1066.639,300.177,-95.789,173.965,32.266,155.914
C03181=1066.645,300.425,-95.821,173.968,32.270,155.915
C03182=1066.651,300.674,-95.853,173.971,32.274,155.916
C03183=1066.657,300.921,-95.884,173.974,32.278,155.917
C03184=1066.663,301.169,-95.916,173.977,32.283,155.917
C03185=1066.670,301.417,-95.948,173.980,32.287,155.918
C03186=1066.675,301.664,-95.980,173.983,32.292,155.919
C03187=1066.682,301.912,-96.012,173.986,32.296,155.920
C03188=1066.688,302.160,-96.044,173.988,32.300,155.921
C03189=1066.694,302.408,-96.076,173.992,32.305,155.922
C03190=1066.699,302.656,-96.107,173.995,32.309,155.922
C03191=1066.706,302.903,-96.139,173.998,32.313,155.923
C03192=1066.712,303.151,-96.171,174.001,32.317,155.924
C03193=1066.718,303.383,-96.201,174.004,32.322,155.925
C03194=1066.723,303.613,-96.231,174.007,32.325,155.925
C03195=1066.730,303.844,-96.261,174.010,32.330,155.926
C03196=1066.735,304.075,-96.291,174.012,32.333,155.927
C03197=1066.741,304.306,-96.320,174.015,32.337,155.928
C03198=1066.746,304.537,-96.350,174.017,32.342,155.929
C03199=1066.752,304.768,-96.380,174.020,32.345,155.929
C03200=1066.758,304.999,-96.411,174.023,32.350,155.930
C03201=1066.765,305.247,-96.442,174.026,32.354,155.931
C03202=1066.770,305.494,-96.475,174.029,32.358,155.932
C03203=1066.776,305.742,-96.507,174.033,32.363,155.932
C03204=1066.782,305.990,-96.539,174.036,32.367,155.933
C03205=1066.788,306.238,-96.571,174.039,32.371,155.934
C03206=1066.795,306.486,-96.603,174.042,32.375,155.935
C03207=1066.802,306.733,-96.636,174.045,32.380,155.936
C03208=1066.808,306.981,-96.668,174.048,32.384,155.937
C03209=1066.814,307.229,-96.700,174.051,32.389,155.937
C03210=1066.819,307.477,-96.732,174.054,32.393,155.938
C03211=1066.826,307.724,-96.764,174.057,32.397,155.939
C03212=1066.832,307.972,-96.796,174.060,32.401,155.940
C03213=1066.838,308.220,-96.829,174.063,32.406,155.941
C03214=1066.844,308.468,-96.861,174.066,32.410,155.942
C03215=1066.851,308.715,-96.894,174.069,32.415,155.942
C03216=1066.857,308.963,-96.926,174.073,32.419,155.943
C03217=1066.863,309.211,-96.958,174.076,32.423,155.944
C03218=1066.870,309.459,-96.991,174.079,32.428,155.945
C03219=1066.876,309.707,-97.023,174.082,32.432,155.946
C03220=1066.882,309.954,-97.055,174.085,32.436,155.946
C03221=1066.889,310.202,-97.088,174.088,32.441,155.947
C03222=1066.895,310.450,-97.120,174.091,32.445,155.948
C03223=1066.901,310.698,-97.153,174.094,32.449,155.949
C03224=1066.907,310.945,-97.186,174.097,32.454,155.950
C03225=1066.914,311.193,-97.218,174.100,32.458,155.951
C03226=1066.920,311.441,-97.250,174.104,32.463,155.951
C03227=1066.927,311.689,-97.283,174.107,32.467,155.952
C03228=1066.933,311.937,-97.316,174.110,32.471,155.953
C03229=1066.940,312.184,-97.348,174.113,32.475,155.954
C03230=1066.946,312.432,-97.381,174.117,32.480,155.955
C03231=1066.952,312.680,-97.413,174.120,32.485,155.956
C03232=1066.958,312.928,-97.446,174.123,32.489,155.956
C03233=1066.965,313.175,-97.479,174.126,32.493,155.957
C03234=1066.971,313.423,-97.511,174.129,32.497,155.958
C03235=1066.978,313.671,-97.544,174.132,32.502,155.959
C03236=1066.984,313.919,-97.577,174.135,32.506,155.960
C03237=1066.990,314.166,-97.610,174.138,32.511,155.961
C03238=1066.997,314.414,-97.643,174.141,32.515,155.961
C03239=1067.003,314.662,-97.675,174.145,32.520,155.962
C03240=1067.009,314.909,-97.709,174.148,32.525,155.963
C03241=1067.015,315.157,-97.742,174.151,32.529,155.964
C03242=1067.020,315.405,-97.775,174.154,32.534,155.965
C03243=1067.027,315.653,-97.808,174.158,32.538,155.966
C03244=1067.033,315.900,-97.840,174.161,32.543,155.967
C03245=1067.038,316.148,-97.874,174.164,32.547,155.967
C03246=1067.045,316.396,-97.906,174.167,32.552,155.968
C03247=1067.051,316.644,-97.940,174.170,32.556,155.969
C03248=1067.058,316.891,-97.974,174.174,32.561,155.970
C03249=1067.063,317.124,-98.005,174.177,32.565,155.971
C03250=1067.069,317.357,-98.036,174.179,32.569,155.972
C03251=1067.075,317.589,-98.067,174.182,32.573,155.973
C03252=1067.081,317.822,-98.098,174.185,32.578,155.974
C03253=1067.086,318.055,-98.129,174.188,32.582,155.974
C03254=1067.092,318.288,-98.161,174.191,32.587,155.975
C03255=1067.097,318.520,-98.192,174.194,32.591,155.976
C03256=1067.104,318.753,-98.223,174.197,32.595,155.977
C03257=1067.109,319.001,-98.256,174.201,32.600,155.978
C03258=1067.116,319.248,-98.289,174.204,32.605,155.979
C03259=1067.121,319.496,-98.323,174.207,32.609,155.979
C03260=1067.128,319.744,-98.356,174.210,32.614,155.980
C03261=1067.134,319.991,-98.390,174.214,32.618,155.981
C03262=1067.140,320.239,-98.423,174.217,32.623,155.982
C03263=1067.146,320.486,-98.457,174.220,32.627,155.983
C03264=1067.153,320.735,-98.490,174.224,32.632,155.984
C03265=1067.159,320.983,-98.523,174.227,32.637,155.985
C03266=1067.165,321.229,-98.557,174.230,32.641,155.986
C03267=1067.171,321.478,-98.590,174.233,32.645,155.987
C03268=1067.178,321.725,-98.624,174.237,32.650,155.987
C03269=1067.183,321.973,-98.657,174.240,32.655,155.988
C03270=1067.190,322.220,-98.691,174.242,32.660,155.989
C03271=1067.196,322.469,-98.724,174.246,32.664,155.990
C03272=1067.203,322.716,-98.758,174.249,32.669,155.991
C03273=1067.209,322.964,-98.791,174.252,32.674,155.992
C03274=1067.216,323.211,-98.825,174.256,32.678,155.993
C03275=1067.221,323.459,-98.858,174.259,32.683,155.994
C03276=1067.228,323.707,-98.892,174.262,32.687,155.995
C03277=1067.234,323.954,-98.926,174.266,32.692,155.996
C03278=1067.240,324.202,-98.959,174.269,32.697,155.996
C03279=1067.247,324.450,-98.993,174.272,32.701,155.997
C03280=1067.253,324.697,-99.027,174.276,32.706,155.998
C03281=1067.260,324.945,-99.060,174.279,32.711,155.999
C03282=1067.266,325.192,-99.094,174.283,32.716,156.000
C03283=1067.273,325.440,-99.128,174.286,32.720,156.001
C03284=1067.278,325.688,-99.162,174.289,32.725,156.002
C03285=1067.285,325.935,-99.195,174.293,32.730,156.003
C03286=1067.291,326.183,-99.229,174.296,32.734,156.004
C03287=1067.297,326.430,-99.264,174.299,32.739,156.005
C03288=1067.304,326.678,-99.297,174.303,32.743,156.006
C03289=1067.310,326.926,-99.331,174.306,32.748,156.007
C03290=1067.317,327.173,-99.365,174.310,32.753,156.007
C03291=1067.323,327.421,-99.399,174.313,32.758,156.008
C03292=1067.330,327.669,-99.433,174.316,32.762,156.009
C03293=1067.337,327.916,-99.467,174.320,32.767,156.010
C03294=1067.343,328.164,-99.501,174.323,32.772,156.011
C03295=1067.350,328.411,-99.535,174.327,32.776,156.012
C03296=1067.355,328.659,-99.568,174.330,32.781,156.013
C03297=1067.362,328.907,-99.602,174.333,32.786,156.014
C03298=1067.368,329.154,-99.636,174.336,32.791,156.015
C03299=1067.375,329.402,-99.670,174.339,32.795,156.016
C03300=1067.381,329.650,-99.705,174.343,32.800,156.017
C03301=1067.388,329.897,-99.738,174.346,32.805,156.018
C03302=1067.394,330.145,-99.773,174.350,32.810,156.019
C03303=1067.400,330.392,-99.807,174.353,32.814,156.020
C03304=1067.407,330.640,-99.841,174.357,32.819,156.020
C03305=1067.414,330.870,-99.873,174.360,32.823,156.021
C03306=1067.420,331.100,-99.904,174.363,32.828,156.022
C03307=1067.426,331.329,-99.936,174.366,32.832,156.023
C03308=1067.431,331.559,-99.968,174.369,32.837,156.024
C03309=1067.437,331.789,-100.001,174.373,32.841,156.025
C03310=1067.443,332.018,-100.032,174.376,32.846,156.026
C03311=1067.449,332.248,-100.064,174.379,32.851,156.027
C03312=1067.455,332.478,-100.096,174.382,32.855,156.027
C03313=1067.461,332.725,-100.130,174.386,32.860,156.029
C03314=1067.467,332.973,-100.165,174.389,32.865,156.029
C03315=1067.473,333.220,-100.199,174.392,32.870,156.030
C03316=1067.480,333.468,-100.233,174.396,32.875,156.031
C03317=1067.487,333.715,-100.269,174.399,32.880,156.032
C03318=1067.492,333.962,-100.303,174.403,32.885,156.033
C03319=1067.499,334.210,-100.337,174.406,32.889,156.034
C03320=1067.506,334.458,-100.372,174.410,32.894,156.035
C03321=1067.512,334.705,-100.406,174.413,32.899,156.036
C03322=1067.518,334.952,-100.441,174.417,32.904,156.037
C03323=1067.525,335.200,-100.476,174.420,32.909,156.038
C03324=1067.530,335.447,-100.511,174.424,32.914,156.039
C03325=1067.537,335.695,-100.546,174.427,32.919,156.040
C03326=1067.543,335.943,-100.580,174.431,32.924,156.041
C03327=1067.550,336.191,-100.615,174.434,32.929,156.042
C03328=1067.556,336.437,-100.650,174.438,32.934,156.043
C03329=1067.563,336.685,-100.684,174.441,32.939,156.044
C03330=1067.569,336.933,-100.719,174.445,32.944,156.045
C03331=1067.576,337.181,-100.754,174.448,32.949,156.046
C03332=1067.583,337.428,-100.789,174.452,32.954,156.047
C03333=1067.588,337.675,-100.823,174.456,32.959,156.048
C03334=1067.594,337.923,-100.859,174.459,32.964,156.049
C03335=1067.601,338.170,-100.894,174.463,32.969,156.050
C03336=1067.608,338.418,-100.928,174.466,32.974,156.051
C03337=1067.614,338.665,-100.963,174.470,32.979,156.052
C03338=1067.620,338.913,-100.999,174.473,32.984,156.053
C03339=1067.627,339.160,-101.034,174.477,32.990,156.054
C03340=1067.633,339.408,-101.068,174.480,32.994,156.055
C03341=1067.639,339.656,-101.104,174.484,33.000,156.056
C03342=1067.646,339.903,-101.139,174.487,33.005,156.057
C03343=1067.652,340.150,-101.174,174.491,33.010,156.058
C03344=1067.659,340.397,-101.209,174.495,33.015,156.059
C03345=1067.665,340.645,-101.244,174.498,33.020,156.060
C03346=1067.671,340.893,-101.279,174.502,33.025,156.061
C03347=1067.678,341.140,-101.314,174.505,33.030,156.062
C03348=1067.684,341.388,-101.350,174.509,33.036,156.063
C03349=1067.691,341.635,-101.385,174.513,33.040,156.064
C03350=1067.698,341.883,-101.420,174.517,33.046,156.065
C03351=1067.703,342.130,-101.456,174.521,33.051,156.067
C03352=1067.710,342.377,-101.491,174.524,33.056,156.068
C03353=1067.717,342.624,-101.526,174.528,33.061,156.069
C03354=1067.723,342.872,-101.562,174.531,33.066,156.070
C03355=1067.729,343.119,-101.597,174.535,33.071,156.071
C03356=1067.736,343.367,-101.632,174.539,33.077,156.072
C03357=1067.742,343.614,-101.668,174.542,33.081,156.073
C03358=1067.749,343.862,-101.703,174.546,33.087,156.074
C03359=1067.755,344.109,-101.739,174.550,33.092,156.075
C03360=1067.762,344.357,-101.774,174.553,33.097,156.076
C03361=1067.767,344.584,-101.807,174.556,33.102,156.077
C03362=1067.774,344.811,-101.840,174.560,33.107,156.078
C03363=1067.779,345.039,-101.872,174.563,33.112,156.079
C03364=1067.786,345.265,-101.905,174.566,33.117,156.080
C03365=1067.791,345.493,-101.937,174.570,33.121,156.081
C03366=1067.798,345.720,-101.970,174.573,33.127,156.082
C03367=1067.803,345.947,-102.003,174.577,33.131,156.083
C03368=1067.809,346.175,-102.036,174.580,33.136,156.084
C03369=1067.816,346.421,-102.071,174.584,33.141,156.085
C03370=1067.822,346.669,-102.107,174.587,33.147,156.086
C03371=1067.828,346.917,-102.143,174.591,33.152,156.087
C03372=1067.835,347.163,-102.179,174.594,33.157,156.088
C03373=1067.841,347.411,-102.214,174.598,33.163,156.089
C03374=1067.848,347.658,-102.250,174.602,33.168,156.090
C03375=1067.854,347.906,-102.286,174.607,33.174,156.091
C03376=1067.861,348.153,-102.323,174.610,33.179,156.092
C03377=1067.868,348.401,-102.358,174.614,33.184,156.094
C03378=1067.874,348.648,-102.394,174.618,33.190,156.095
C03379=1067.880,348.895,-102.430,174.621,33.195,156.096
C03380=1067.887,349.142,-102.466,174.625,33.201,156.097
C03381=1067.893,349.390,-102.502,174.629,33.206,156.098
C03382=1067.900,349.637,-102.538,174.632,33.211,156.099
C03383=1067.906,349.885,-102.574,174.636,33.217,156.100
C03384=1067.913,350.131,-102.610,174.640,33.222,156.101
C03385=1067.919,350.380,-102.646,174.644,33.228,156.102
C03386=1067.926,350.627,-102.682,174.647,33.233,156.104
C03387=1067.933,350.874,-102.718,174.651,33.239,156.105
C03388=1067.939,351.121,-102.754,174.655,33.244,156.106
C03389=1067.945,351.368,-102.790,174.658,33.250,156.107
C03390=1067.952,351.616,-102.827,174.663,33.255,156.108
C03391=1067.959,351.863,-102.863,174.667,33.260,156.109
C03392=1067.965,352.110,-102.899,174.671,33.266,156.110
C03393=1067.971,352.357,-102.935,174.674,33.271,156.111
C03394=1067.978,352.605,-102.972,174.678,33.277,156.113
C03395=1067.985,352.852,-103.008,174.682,33.282,156.114
C03396=1067.991,353.099,-103.045,174.686,33.288,156.115
C03397=1067.997,353.346,-103.081,174.689,33.293,156.116
C03398=1068.004,353.594,-103.116,174.693,33.299,156.117
C03399=1068.011,353.842,-103.153,174.697,33.305,156.118
C03400=1068.017,354.089,-103.190,174.701,33.310,156.119
C03401=1068.024,354.336,-103.226,174.704,33.316,156.121
C03402=1068.030,354.583,-103.263,174.709,33.322,156.122
C03403=1068.037,354.830,-103.299,174.713,33.327,156.123
C03404=1068.043,355.077,-103.336,174.717,33.333,156.124
C03405=1068.050,355.325,-103.372,174.721,33.339,156.125
C03406=1068.057,355.572,-103.409,174.724,33.344,156.126
C03407=1068.063,355.819,-103.446,174.728,33.350,156.128
C03408=1068.070,356.066,-103.483,174.732,33.356,156.129
C03409=1068.077,356.314,-103.519,174.736,33.361,156.130
C03410=1068.083,356.561,-103.556,174.740,33.367,156.131
C03411=1068.089,356.808,-103.592,174.743,33.372,156.132
C03412=1068.096,357.055,-103.629,174.748,33.378,156.133
C03413=1068.103,357.302,-103.666,174.752,33.384,156.135
C03414=1068.109,357.549,-103.703,174.756,33.390,156.136
C03415=1068.116,357.797,-103.740,174.760,33.396,156.137
C03416=1068.122,358.044,-103.776,174.764,33.401,156.138
C03417=1068.129,358.273,-103.811,174.767,33.407,156.139
C03418=1068.135,358.502,-103.844,174.771,33.412,156.140
C03419=1068.141,358.731,-103.879,174.774,33.417,156.142
C03420=1068.147,358.961,-103.913,174.778,33.422,156.143
C03421=1068.153,359.190,-103.947,174.782,33.428,156.144
C03422=1068.159,359.418,-103.982,174.786,33.433,156.145
C03423=1068.166,359.648,-104.016,174.790,33.439,156.146
C03424=1068.171,359.877,-104.051,174.793,33.444,156.147
C03425=1068.178,360.124,-104.087,174.797,33.450,156.148
C03426=1068.185,360.371,-104.125,174.801,33.456,156.150
C03427=1068.191,360.618,-104.161,174.805,33.461,156.151
C03428=1068.199,360.866,-104.199,174.809,33.467,156.152
C03429=1068.204,361.112,-104.236,174.813,33.474,156.153
C03430=1068.211,361.360,-104.273,174.817,33.479,156.155
C03431=1068.218,361.606,-104.310,174.821,33.485,156.156
C03432=1068.225,361.854,-104.347,174.825,33.491,156.157
C03433=1068.232,362.101,-104.384,174.829,33.497,156.158
C03434=1068.238,362.348,-104.422,174.833,33.503,156.160
C03435=1068.245,362.595,-104.459,174.837,33.509,156.161
C03436=1068.252,362.842,-104.496,174.841,33.515,156.162
C03437=1068.258,363.089,-104.533,174.846,33.521,156.163
C03438=1068.265,363.337,-104.571,174.850,33.527,156.164
C03439=1068.272,363.584,-104.608,174.854,33.533,156.166
C03440=1068.278,363.830,-104.646,174.858,33.539,156.167
C03441=1068.285,364.078,-104.684,174.861,33.545,156.168
C03442=1068.292,364.324,-104.721,174.865,33.551,156.170
C03443=1068.299,364.572,-104.758,174.870,33.557,156.171
C03444=1068.305,364.819,-104.796,174.874,33.563,156.172
C03445=1068.312,365.066,-104.833,174.878,33.569,156.173
C03446=1068.318,365.313,-104.871,174.882,33.575,156.175
C03447=1068.325,365.560,-104.908,174.886,33.581,156.176
C03448=1068.331,365.807,-104.946,174.890,33.587,156.177
C03449=1068.339,366.054,-104.984,174.895,33.594,156.179
C03450=1068.345,366.301,-105.022,174.899,33.600,156.180
C03451=1068.352,366.548,-105.059,174.903,33.606,156.181
C03452=1068.358,366.796,-105.097,174.907,33.612,156.183
C03453=1068.364,367.042,-105.135,174.911,33.618,156.184
C03454=1068.371,367.290,-105.173,174.915,33.624,156.185
C03455=1068.378,367.536,-105.211,174.920,33.630,156.186
C03456=1068.385,367.783,-105.249,174.924,33.637,156.188
C03457=1068.391,368.030,-105.287,174.928,33.643,156.189
C03458=1068.399,368.277,-105.324,174.932,33.649,156.190
C03459=1068.405,368.524,-105.362,174.936,33.656,156.192
C03460=1068.412,368.771,-105.400,174.940,33.662,156.193
C03461=1068.419,369.018,-105.438,174.945,33.668,156.194
C03462=1068.425,369.266,-105.476,174.949,33.674,156.196
C03463=1068.432,369.513,-105.514,174.953,33.681,156.197
C03464=1068.439,369.759,-105.552,174.957,33.687,156.199
C03465=1068.446,370.006,-105.590,174.961,33.693,156.200
C03466=1068.452,370.253,-105.628,174.966,33.700,156.201
C03467=1068.459,370.500,-105.667,174.970,33.706,156.203
C03468=1068.466,370.747,-105.704,174.974,33.712,156.204
C03469=1068.473,370.993,-105.743,174.978,33.718,156.205
C03470=1068.480,371.241,-105.780,174.982,33.725,156.207
C03471=1068.487,371.487,-105.819,174.987,33.731,156.208
C03472=1068.493,371.735,-105.857,174.991,33.738,156.209
C03473=1068.500,371.973,-105.894,174.995,33.743,156.211
C03474=1068.506,372.210,-105.931,174.999,33.750,156.212
C03475=1068.513,372.448,-105.968,175.004,33.756,156.213
C03476=1068.520,372.686,-106.005,175.008,33.762,156.215
C03477=1068.526,372.923,-106.041,175.012,33.769,156.216
C03478=1068.533,373.161,-106.079,175.016,33.775,156.217
C03479=1068.539,373.399,-106.116,175.020,33.781,156.219
C03480=1068.546,373.637,-106.153,175.025,33.787,156.220
C03481=1068.552,373.883,-106.191,175.029,33.794,156.221
C03482=1068.559,374.130,-106.230,175.033,33.800,156.223
C03483=1068.566,374.377,-106.269,175.037,33.807,156.224
C03484=1068.573,374.624,-106.307,175.042,33.814,156.226
C03485=1068.579,374.871,-106.346,175.047,33.820,156.227
C03486=1068.586,375.118,-106.385,175.051,33.827,156.229
C03487=1068.593,375.365,-106.424,175.055,33.834,156.230
C03488=1068.601,375.611,-106.462,175.060,33.840,156.231
C03489=1068.607,375.858,-106.501,175.064,33.847,156.233
C03490=1068.614,376.105,-106.539,175.068,33.854,156.234
C03491=1068.621,376.352,-106.578,175.072,33.860,156.236
C03492=1068.628,376.599,-106.617,175.077,33.867,156.237
C03493=1068.635,376.845,-106.656,175.082,33.874,156.239
C03494=1068.641,377.092,-106.695,175.086,33.880,156.240
C03495=1068.648,377.339,-106.734,175.090,33.887,156.242
C03496=1068.655,377.586,-106.772,175.095,33.894,156.243
C03497=1068.662,377.833,-106.811,175.099,33.901,156.245
C03498=1068.669,378.079,-106.850,175.104,33.907,156.246
C03499=1068.675,378.326,-106.889,175.108,33.914,156.248
C03500=1068.682,378.573,-106.928,175.113,33.921,156.249
C03501=1068.690,378.820,-106.968,175.117,33.928,156.250
C03502=1068.697,379.067,-107.007,175.121,33.935,156.252
C03503=1068.704,379.314,-107.045,175.127,33.941,156.253
C03504=1068.710,379.561,-107.084,175.131,33.948,156.255
C03505=1068.718,379.807,-107.124,175.135,33.955,156.256
C03506=1068.724,380.054,-107.163,175.139,33.962,156.258
C03507=1068.731,380.300,-107.201,175.144,33.969,156.259
C03508=1068.739,380.547,-107.241,175.149,33.976,156.261
C03509=1068.746,380.794,-107.280,175.153,33.982,156.262
C03510=1068.753,381.041,-107.319,175.158,33.990,156.264
C03511=1068.760,381.287,-107.359,175.162,33.997,156.266
C03512=1068.766,381.535,-107.398,175.167,34.003,156.267
C03513=1068.773,381.781,-107.438,175.172,34.011,156.269
C03514=1068.780,382.028,-107.477,175.176,34.017,156.270
C03515=1068.787,382.274,-107.516,175.181,34.025,156.272
C03516=1068.794,382.521,-107.556,175.186,34.032,156.273
C03517=1068.801,382.768,-107.596,175.190,34.039,156.275
C03518=1068.808,383.014,-107.635,175.194,34.046,156.276
C03519=1068.815,383.261,-107.675,175.200,34.053,156.278
C03520=1068.821,383.508,-107.714,175.204,34.060,156.279
C03521=1068.829,383.755,-107.754,175.208,34.067,156.281
C03522=1068.836,384.001,-107.794,175.213,34.075,156.283
C03523=1068.842,384.248,-107.833,175.218,34.082,156.284
C03524=1068.849,384.495,-107.873,175.222,34.089,156.286
C03525=1068.857,384.741,-107.913,175.227,34.096,156.287
C03526=1068.864,384.988,-107.953,175.232,34.103,156.289
C03527=1068.870,385.234,-107.993,175.236,34.110,156.291
C03528=1068.878,385.481,-108.033,175.241,34.118,156.292
C03529=1068.884,385.713,-108.070,175.246,34.125,156.294
C03530=1068.891,385.947,-108.108,175.250,34.132,156.295
C03531=1068.897,386.180,-108.145,175.255,34.138,156.297
C03532=1068.904,386.413,-108.183,175.259,34.145,156.298
C03533=1068.911,386.645,-108.221,175.263,34.152,156.300
C03534=1068.917,386.878,-108.259,175.268,34.159,156.301
C03535=1068.924,387.111,-108.296,175.272,34.166,156.303
C03536=1068.931,387.344,-108.334,175.276,34.173,156.305
C03537=1068.938,387.590,-108.374,175.282,34.180,156.306
C03538=1068.945,387.837,-108.414,175.286,34.188,156.308
C03539=1068.952,388.083,-108.454,175.292,34.195,156.310
C03540=1068.959,388.330,-108.495,175.296,34.203,156.311
C03541=1068.966,388.576,-108.534,175.300,34.210,156.313
C03542=1068.973,388.823,-108.575,175.306,34.218,156.314
C03543=1068.981,389.070,-108.614,175.310,34.225,156.316
C03544=1068.989,389.316,-108.655,175.316,34.233,156.318
C03545=1068.996,389.563,-108.696,175.320,34.240,156.319
C03546=1069.003,389.809,-108.735,175.325,34.248,156.321
C03547=1069.010,390.056,-108.776,175.330,34.255,156.323
C03548=1069.017,390.302,-108.816,175.335,34.263,156.325
C03549=1069.024,390.549,-108.856,175.340,34.270,156.326
C03550=1069.032,390.796,-108.897,175.345,34.278,156.328
C03551=1069.038,391.042,-108.937,175.350,34.286,156.330
C03552=1069.046,391.289,-108.978,175.354,34.293,156.331
C03553=1069.053,391.535,-109.018,175.359,34.301,156.333
C03554=1069.060,391.781,-109.059,175.364,34.309,156.335
C03555=1069.067,392.029,-109.100,175.369,34.316,156.337
C03556=1069.075,392.274,-109.140,175.374,34.324,156.338
C03557=1069.082,392.521,-109.181,175.379,34.332,156.340
C03558=1069.088,392.767,-109.221,175.384,34.339,156.342
C03559=1069.096,393.014,-109.263,175.389,34.348,156.344
C03560=1069.104,393.260,-109.303,175.395,34.356,156.345
C03561=1069.111,393.507,-109.344,175.399,34.363,156.347
C03562=1069.117,393.753,-109.385,175.405,34.371,156.349
C03563=1069.125,394.000,-109.426,175.409,34.379,156.351
C03564=1069.133,394.246,-109.466,175.415,34.387,156.352
C03565=1069.140,394.493,-109.508,175.419,34.395,156.354
C03566=1069.146,394.739,-109.548,175.424,34.403,156.356
C03567=1069.154,394.986,-109.589,175.429,34.411,156.358
C03568=1069.161,395.233,-109.630,175.434,34.419,156.360
C03569=1069.168,395.479,-109.672,175.439,34.427,156.362
C03570=1069.175,395.725,-109.712,175.444,34.435,156.363
C03571=1069.182,395.972,-109.754,175.450,34.443,156.365
C03572=1069.189,396.218,-109.795,175.455,34.451,156.367
C03573=1069.197,396.465,-109.836,175.460,34.459,156.369
C03574=1069.205,396.711,-109.877,175.465,34.467,156.371
C03575=1069.212,396.957,-109.919,175.470,34.475,156.373
C03576=1069.220,397.204,-109.960,175.476,34.483,156.374
C03577=1069.227,397.450,-110.001,175.480,34.491,156.376
C03578=1069.234,397.697,-110.042,175.486,34.500,156.378
C03579=1069.241,397.943,-110.084,175.490,34.508,156.380
C03580=1069.248,398.189,-110.124,175.496,34.516,156.382
C03581=1069.257,398.476,-110.173,175.501,34.526,156.384
C03582=1069.265,398.761,-110.222,175.508,34.536,156.386
C03583=1069.274,399.047,-110.269,175.514,34.545,156.389
C03584=1069.282,399.334,-110.318,175.520,34.555,156.391
C03585=1069.291,399.608,-110.364,175.526,34.564,156.393
C03586=1069.298,399.882,-110.411,175.532,34.573,156.395
C03587=1069.307,400.158,-110.457,175.537,34.583,156.397
C03588=1069.315,400.431,-110.504,175.544,34.592,156.399
C03589=1069.322,400.678,-110.545,175.549,34.600,156.401
C03590=1069.329,400.924,-110.587,175.554,34.609,156.403
C03591=1069.337,401.171,-110.629,175.560,34.617,156.405
C03592=1069.345,401.418,-110.671,175.564,34.626,156.407
C03593=1069.352,401.664,-110.712,175.570,34.634,156.409
C03594=1069.360,401.910,-110.754,175.576,34.643,156.411
C03595=1069.366,402.156,-110.797,175.581,34.652,156.413
C03596=1069.374,402.403,-110.838,175.586,34.660,156.415
C03597=1069.381,402.649,-110.880,175.591,34.669,156.417
C03598=1069.390,402.896,-110.922,175.597,34.678,156.419
C03599=1069.396,403.142,-110.965,175.603,34.686,156.421
C03600=1069.404,403.388,-111.007,175.607,34.695,156.423
C03601=1069.412,403.634,-111.049,175.613,34.704,156.425
C03602=1069.418,403.881,-111.090,175.619,34.713,156.427
C03603=1069.426,404.127,-111.133,175.624,34.721,156.429
C03604=1069.434,404.373,-111.175,175.630,34.730,156.431
C03605=1069.441,404.620,-111.217,175.636,34.739,156.433
C03606=1069.449,404.866,-111.260,175.640,34.747,156.435
C03607=1069.457,405.112,-111.302,175.646,34.756,156.437
C03608=1069.464,405.358,-111.345,175.652,34.765,156.440
C03609=1069.471,405.604,-111.387,175.657,34.774,156.442
C03610=1069.479,405.851,-111.430,175.663,34.783,156.444
C03611=1069.486,406.097,-111.472,175.669,34.792,156.446
C03612=1069.494,406.344,-111.514,175.674,34.801,156.448
C03613=1069.501,406.590,-111.556,175.679,34.810,156.450
C03614=1069.509,406.836,-111.600,175.685,34.819,156.452
C03615=1069.516,407.083,-111.643,175.691,34.829,156.454
C03616=1069.524,407.329,-111.685,175.696,34.837,156.456
C03617=1069.531,407.574,-111.728,175.702,34.847,156.459
C03618=1069.539,407.821,-111.770,175.708,34.856,156.461
C03619=1069.546,408.067,-111.813,175.714,34.865,156.463
C03620=1069.554,408.314,-111.856,175.719,34.874,156.465
C03621=1069.561,408.560,-111.898,175.725,34.883,156.467
C03622=1069.569,408.806,-111.942,175.731,34.893,156.469
C03623=1069.576,409.052,-111.985,175.737,34.902,156.472
C03624=1069.584,409.298,-112.027,175.742,34.911,156.474
C03625=1069.591,409.544,-112.071,175.748,34.921,156.476
C03626=1069.599,409.791,-112.114,175.754,34.930,156.478
C03627=1069.607,410.036,-112.156,175.760,34.939,156.480
C03628=1069.615,410.283,-112.200,175.766,34.949,156.483
C03629=1069.621,410.529,-112.242,175.771,34.958,156.485
C03630=1069.629,410.775,-112.286,175.777,34.967,156.487
C03631=1069.638,411.021,-112.329,175.783,34.977,156.489
C03632=1069.645,411.267,-112.372,175.789,34.986,156.492
C03633=1069.653,411.513,-112.416,175.795,34.996,156.494
